    LOCAL CONST Robtarget Tr_meulage_bavure_392 := [[123.2293125,134.237953125,21.5],[0.365324878383577,-0.417802676522739,-0.626220329354095,0.547564385098326],[0,0,0,0],[8.999999E+09,8.999999E+09,8.999999E+09,8.999999E+09,8.999999E+09,8.999999E+09]];
    LOCAL CONST Robtarget Tr_meulage_bavure_393 := [[120.6318984375,139.860234375,21.5],[0.3646126685295,-0.41742546939904,-0.626882481156863,0.547569113686486],[0,0,0,0],[8.999999E+09,8.999999E+09,8.999999E+09,8.999999E+09,8.999999E+09,8.999999E+09]];
    LOCAL CONST Robtarget Tr_meulage_bavure_394 := [[119.7307734375,142.1045,21.5],[0.363803096049032,-0.416925869952999,-0.627615947970583,0.547648014807011],[0,0,0,0],[8.999999E+09,8.999999E+09,8.999999E+09,8.999999E+09,8.999999E+09,8.999999E+09]];
    LOCAL CONST Robtarget Tr_meulage_bavure_395 := [[119.108765625,144.030703125,21.5],[0.362728439124589,-0.416118032571449,-0.628549716058463,0.547904295349043],[0,0,0,0],[8.999999E+09,8.999999E+09,8.999999E+09,8.999999E+09,8.999999E+09,8.999999E+09]];
    LOCAL CONST Robtarget Tr_meulage_bavure_396 := [[118.348453125,146.077265625,21.5],[0.361294289455634,-0.414888689677899,-0.629752649770469,0.548402600004028],[0,0,0,0],[8.999999E+09,8.999999E+09,8.999999E+09,8.999999E+09,8.999999E+09,8.999999E+09]];
    LOCAL CONST Robtarget Tr_meulage_bavure_397 := [[117.2526875,148.617953125,21.5],[0.35949752433227,-0.413236866055573,-0.631224964075012,0.549137384686234],[0,0,0,0],[8.999999E+09,8.999999E+09,8.999999E+09,8.999999E+09,8.999999E+09,8.999999E+09]];
    LOCAL CONST Robtarget Tr_meulage_bavure_398 := [[116.4586171875,150.514953125,21.5],[0.357426668393585,-0.411263124366953,-0.632896063989253,0.550046717510346],[0,0,0,0],[8.999999E+09,8.999999E+09,8.999999E+09,8.999999E+09,8.999999E+09,8.999999E+09]];
    LOCAL CONST Robtarget Tr_meulage_bavure_399 := [[115.483578125,152.6576875,21.5],[0.355235316197575,-0.409147915918491,-0.634649279253162,0.55102281746676],[0,0,0,0],[8.999999E+09,8.999999E+09,8.999999E+09,8.999999E+09,8.999999E+09,8.999999E+09]];
    LOCAL CONST Robtarget Tr_meulage_bavure_400 := [[115.30321875,153.038,21.5],[0.353116300669102,-0.407109354480308,-0.636339473739805,0.551944676445876],[0,0,0,0],[8.999999E+09,8.999999E+09,8.999999E+09,8.999999E+09,8.999999E+09,8.999999E+09]];
    LOCAL CONST Robtarget Tr_meulage_bavure_401 := [[113.392453125,157.026609375,21.5],[0.351249562294065,-0.405358318756695,-0.637836707518237,0.552695859352383],[0,0,0,0],[8.999999E+09,8.999999E+09,8.999999E+09,8.999999E+09,8.999999E+09,8.999999E+09]];
    LOCAL CONST Robtarget Tr_meulage_bavure_402 := [[111.789640625,160.5481875,21.5],[0.349780045613179,-0.404061741909902,-0.639037894404603,0.553189477422075],[0,0,0,0],[8.999999E+09,8.999999E+09,8.999999E+09,8.999999E+09,8.999999E+09,8.999999E+09]];
    LOCAL CONST Robtarget Tr_meulage_bavure_403 := [[111.554078125,161.02996875,21.5],[0.348771840415515,-0.403295967871138,-0.639900183230376,0.553388038480945],[0,0,0,0],[8.999999E+09,8.999999E+09,8.999999E+09,8.999999E+09,8.999999E+09,8.999999E+09]];
    LOCAL CONST Robtarget Tr_meulage_bavure_404 := [[111.5132421875,161.124546875,21.5],[0.348208503244956,-0.403042649721828,-0.640437546956707,0.553305710454167],[0,0,0,0],[8.999999E+09,8.999999E+09,8.999999E+09,8.999999E+09,8.999999E+09,8.999999E+09]];
    LOCAL CONST Robtarget Tr_meulage_bavure_405 := [[111.45303125,161.24990625,21.5],[0.34797926768379,-0.40317690822812,-0.640731836832706,0.553011322852303],[0,0,0,0],[8.999999E+09,8.999999E+09,8.999999E+09,8.999999E+09,8.999999E+09,8.999999E+09]];
    LOCAL CONST Robtarget Tr_meulage_bavure_406 := [[109.664703125,164.673953125,21.5],[0.347911501640597,-0.40349693803522,-0.640907643054192,0.552616685503711],[0,0,0,0],[8.999999E+09,8.999999E+09,8.999999E+09,8.999999E+09,8.999999E+09,8.999999E+09]];
    LOCAL CONST Robtarget Tr_meulage_bavure_407 := [[109.3512578125,165.311765625,21.5],[0.347796802264797,-0.40375948552209,-0.641116279922809,0.552254993461587],[0,0,0,0],[8.999999E+09,8.999999E+09,8.999999E+09,8.999999E+09,8.999999E+09,8.999999E+09]];
    LOCAL CONST Robtarget Tr_meulage_bavure_408 := [[106.2381875,171.797703125,21.5],[0.347430621451574,-0.403728519395173,-0.641508118263495,0.552053059140862],[0,0,0,0],[8.999999E+09,8.999999E+09,8.999999E+09,8.999999E+09,8.999999E+09,8.999999E+09]];
    LOCAL CONST Robtarget Tr_meulage_bavure_409 := [[105.573640625,173.400671875,21.5],[0.34666342359124,-0.403226194397503,-0.64219160057769,0.552107829181196],[0,0,0,0],[8.999999E+09,8.999999E+09,8.999999E+09,8.999999E+09,8.999999E+09,8.999999E+09]];
    LOCAL CONST Robtarget Tr_meulage_bavure_410 := [[104.5446484375,175.74321875,21.5],[0.345413274544686,-0.402154478934636,-0.643224767495469,0.552470219397869],[0,0,0,0],[8.999999E+09,8.999999E+09,8.999999E+09,8.999999E+09,8.999999E+09,8.999999E+09]];
    LOCAL CONST Robtarget Tr_meulage_bavure_411 := [[103.92953125,176.899171875,21.5],[0.34368116327913,-0.400511497135502,-0.644602879657129,0.553137348410971],[0,0,0,0],[8.999999E+09,8.999999E+09,8.999999E+09,8.999999E+09,8.999999E+09,8.999999E+09]];
    LOCAL CONST Robtarget Tr_meulage_bavure_412 := [[103.241484375,178.22771875,21.5],[0.341551514127714,-0.398394425670201,-0.646259664142013,0.554051343554936],[0,0,0,0],[8.999999E+09,8.999999E+09,8.999999E+09,8.999999E+09,8.999999E+09,8.999999E+09]];
    LOCAL CONST Robtarget Tr_meulage_bavure_413 := [[102.9495859375,178.82403125,21.5],[0.339159708641225,-0.395957401256905,-0.648091582916801,0.555126768023911],[0,0,0,0],[8.999999E+09,8.999999E+09,8.999999E+09,8.999999E+09,8.999999E+09,8.999999E+09]];
    LOCAL CONST Robtarget Tr_meulage_bavure_414 := [[99.8190625,184.99203125,21.5],[0.336664877214233,-0.39338158108794,-0.649980010542665,0.556267631636098],[0,0,0,0],[8.999999E+09,8.999999E+09,8.999999E+09,8.999999E+09,8.999999E+09,8.999999E+09]];
    LOCAL CONST Robtarget Tr_meulage_bavure_415 := [[98.8109765625,186.739015625,21.5],[0.334213643527929,-0.390838206503484,-0.651820001777444,0.557384447307044],[0,0,0,0],[8.999999E+09,8.999999E+09,8.999999E+09,8.999999E+09,8.999999E+09,8.999999E+09]];
    LOCAL CONST Robtarget Tr_meulage_bavure_416 := [[96.223203125,191.122984375,21.5],[0.331906128976775,-0.388441424497442,-0.653541237438173,0.558422270553237],[0,0,0,0],[8.999999E+09,8.999999E+09,8.999999E+09,8.999999E+09,8.999999E+09,8.999999E+09]];
    LOCAL CONST Robtarget Tr_meulage_bavure_417 := [[95.8459453125,191.848875,21.5],[0.329782886774544,-0.386237077058502,-0.655116976082171,0.559362061231279],[0,0,0,0],[8.999999E+09,8.999999E+09,8.999999E+09,8.999999E+09,8.999999E+09,8.999999E+09]];
    LOCAL CONST Robtarget Tr_meulage_bavure_418 := [[92.463046875,198.07146875,21.5],[0.327832239999258,-0.384211623196163,-0.656557507184878,0.560213968745172],[0,0,0,0],[8.999999E+09,8.999999E+09,8.999999E+09,8.999999E+09,8.999999E+09,8.999999E+09]];
    LOCAL CONST Robtarget Tr_meulage_bavure_419 := [[90.7008046875,201.166375,21.5],[0.326001741527339,-0.38230075368062,-0.657899339305977,0.561014667898382],[0,0,0,0],[8.999999E+09,8.999999E+09,8.999999E+09,8.999999E+09,8.999999E+09,8.999999E+09]];
    LOCAL CONST Robtarget Tr_meulage_bavure_420 := [[89.685421875,203.134609375,21.5],[0.32421441231465,-0.380410965519129,-0.659194370838049,0.561814287479145],[0,0,0,0],[8.999999E+09,8.999999E+09,8.999999E+09,8.999999E+09,8.999999E+09,8.999999E+09]];
    LOCAL CONST Robtarget Tr_meulage_bavure_421 := [[88.7899140625,204.7486875,21.5],[0.322389107164825,-0.378447015897074,-0.660497192024121,0.562660269672843],[0,0,0,0],[8.999999E+09,8.999999E+09,8.999999E+09,8.999999E+09,8.999999E+09,8.999999E+09]];
    LOCAL CONST Robtarget Tr_meulage_bavure_422 := [[88.1928984375,205.782015625,21.5],[0.320460920439119,-0.376330604631915,-0.661849248538786,0.563591737605631],[0,0,0,0],[8.999999E+09,8.999999E+09,8.999999E+09,8.999999E+09,8.999999E+09,8.999999E+09]];
    LOCAL CONST Robtarget Tr_meulage_bavure_423 := [[87.51946875,206.94284375,21.5],[0.318384606952656,-0.374006932194033,-0.663277721464299,0.564635033393729],[0,0,0,0],[8.999999E+09,8.999999E+09,8.999999E+09,8.999999E+09,8.999999E+09,8.999999E+09]];
    LOCAL CONST Robtarget Tr_meulage_bavure_424 := [[82.9292265625,214.408875,21.5],[0.316149517900522,-0.371459858394791,-0.664784972159725,0.565798547827036],[0,0,0,0],[8.999999E+09,8.999999E+09,8.999999E+09,8.999999E+09,8.999999E+09,8.999999E+09]];
    LOCAL CONST Robtarget Tr_meulage_bavure_425 := [[82.8541875,214.52709375,21.5],[0.31376219441939,-0.368696993357463,-0.666363021379249,0.567076834459507],[0,0,0,0],[8.999999E+09,8.999999E+09,8.999999E+09,8.999999E+09,8.999999E+09,8.999999E+09]];
    LOCAL CONST Robtarget Tr_meulage_bavure_426 := [[82.726046875,214.73296875,21.5],[0.311250217448688,-0.365749884059349,-0.667989819633394,0.568453978185449],[0,0,0,0],[8.999999E+09,8.999999E+09,8.999999E+09,8.999999E+09,8.999999E+09,8.999999E+09]];
    LOCAL CONST Robtarget Tr_meulage_bavure_427 := [[77.443234375,223.1875625,21.5],[0.308652711768212,-0.362662646255843,-0.669635933625859,0.569909663829156],[0,0,0,0],[8.999999E+09,8.999999E+09,8.999999E+09,8.999999E+09,8.999999E+09,8.999999E+09]];
    LOCAL CONST Robtarget Tr_meulage_bavure_428 := [[76.0887734375,225.3150625,21.5],[0.306016386673545,-0.359491315340013,-0.671269404439817,0.571416968548702],[0,0,0,0],[8.999999E+09,8.999999E+09,8.999999E+09,8.999999E+09,8.999999E+09,8.999999E+09]];
    LOCAL CONST Robtarget Tr_meulage_bavure_429 := [[74.37640625,227.81146875,21.5],[0.303387642067638,-0.356290732601125,-0.672859367913488,0.572951240084402],[0,0,0,0],[8.999999E+09,8.999999E+09,8.999999E+09,8.999999E+09,8.999999E+09,8.999999E+09]];
    LOCAL CONST Robtarget Tr_meulage_bavure_430 := [[68.2574453125,236.729,21.5],[0.300808323404873,-0.353108038227415,-0.674377917318904,0.574494117064877],[0,0,0,0],[8.999999E+09,8.999999E+09,8.999999E+09,8.999999E+09,8.999999E+09,8.999999E+09]];
    LOCAL CONST Robtarget Tr_meulage_bavure_431 := [[67.4715,237.87903125,21.5],[0.298307331372168,-0.349979154564493,-0.675808150496031,0.576030095692119],[0,0,0,0],[8.999999E+09,8.999999E+09,8.999999E+09,8.999999E+09,8.999999E+09,8.999999E+09]];
    LOCAL CONST Robtarget Tr_meulage_bavure_432 := [[64.73254296875,241.804015625,21.5],[0.29590323329365,-0.34692572251121,-0.677139156497948,0.577552060271354],[0,0,0,0],[8.999999E+09,8.999999E+09,8.999999E+09,8.999999E+09,8.999999E+09,8.999999E+09]];
    LOCAL CONST Robtarget Tr_meulage_bavure_433 := [[64.363859375,242.338875,21.5],[0.293608347744609,-0.343964602763721,-0.678365598990462,0.579053196422045],[0,0,0,0],[8.999999E+09,8.999999E+09,8.999999E+09,8.999999E+09,8.999999E+09,8.999999E+09]];
    LOCAL CONST Robtarget Tr_meulage_bavure_434 := [[61.49722265625,246.202390625,21.5],[0.291423878540126,-0.341097438253869,-0.67948788946556,0.580534984908676],[0,0,0,0],[8.999999E+09,8.999999E+09,8.999999E+09,8.999999E+09,8.999999E+09,8.999999E+09]];
    LOCAL CONST Robtarget Tr_meulage_bavure_435 := [[61.4078671875,246.320796875,21.5],[0.289335193516394,-0.338307694283393,-0.680515840627853,0.582006220272646],[0,0,0,0],[8.999999E+09,8.999999E+09,8.999999E+09,8.999999E+09,8.999999E+09,8.999999E+09]];
    LOCAL CONST Robtarget Tr_meulage_bavure_436 := [[60.460328125,247.569390625,21.5],[0.287317708905303,-0.335572671606102,-0.681467718916006,0.583473447807153],[0,0,0,0],[8.999999E+09,8.999999E+09,8.999999E+09,8.999999E+09,8.999999E+09,8.999999E+09]];
    LOCAL CONST Robtarget Tr_meulage_bavure_437 := [[58.3609296875,250.421015625,21.5],[0.285327430113036,-0.332838804964973,-0.682367604268253,0.584962426297437],[0,0,0,0],[8.999999E+09,8.999999E+09,8.999999E+09,8.999999E+09,8.999999E+09,8.999999E+09]];
    LOCAL CONST Robtarget Tr_meulage_bavure_438 := [[56.72735546875,252.611640625,21.5],[0.283294917264907,-0.330032027158558,-0.68325802082939,0.586499213873119],[0,0,0,0],[8.999999E+09,8.999999E+09,8.999999E+09,8.999999E+09,8.999999E+09,8.999999E+09]];
    LOCAL CONST Robtarget Tr_meulage_bavure_439 := [[56.11966015625,253.3434375,21.5],[0.281118816189949,-0.327035188516629,-0.684193876122193,0.588131733995662],[0,0,0,0],[8.999999E+09,8.999999E+09,8.999999E+09,8.999999E+09,8.999999E+09,8.999999E+09]];
    LOCAL CONST Robtarget Tr_meulage_bavure_440 := [[53.942109375,255.9426875,21.5],[0.278670537913217,-0.323704550533762,-0.685244908508551,0.589913138204262],[0,0,0,0],[8.999999E+09,8.999999E+09,8.999999E+09,8.999999E+09,8.999999E+09,8.999999E+09]];
    LOCAL CONST Robtarget Tr_meulage_bavure_441 := [[52.053375,258.2940625,21.5],[0.275780385089803,-0.319847556218044,-0.686497756579809,0.591915154555071],[0,0,0,0],[8.999999E+09,8.999999E+09,8.999999E+09,8.999999E+09,8.999999E+09,8.999999E+09]];
    LOCAL CONST Robtarget Tr_meulage_bavure_442 := [[50.915984375,259.725765625,21.5],[0.272271064189163,-0.315265305626162,-0.688037190555852,0.594206259716064],[0,0,0,0],[8.999999E+09,8.999999E+09,8.999999E+09,8.999999E+09,8.999999E+09,8.999999E+09]];
    LOCAL CONST Robtarget Tr_meulage_bavure_443 := [[50.12555078125,260.70153125,21.5],[0.267918294793822,-0.309709378512022,-0.689965854732275,0.59686431245303],[0,0,0,0],[8.999999E+09,8.999999E+09,8.999999E+09,8.999999E+09,8.999999E+09,8.999999E+09]];
    LOCAL CONST Robtarget Tr_meulage_bavure_444 := [[48.66555859375,262.7159375,21.5],[0.262537588739252,-0.302972431940772,-0.692347864523534,0.599946793034662],[0,0,0,0],[8.999999E+09,8.999999E+09,8.999999E+09,8.999999E+09,8.999999E+09,8.999999E+09]];
    LOCAL CONST Robtarget Tr_meulage_bavure_445 := [[46.71563671875,264.9346875,21.5],[0.255944756105986,-0.29485466848261,-0.695235613162406,0.603490222362012],[0,0,0,0],[8.999999E+09,8.999999E+09,8.999999E+09,8.999999E+09,8.999999E+09,8.999999E+09]];
    LOCAL CONST Robtarget Tr_meulage_bavure_446 := [[46.5646953125,265.1093125,21.5],[0.247999035077578,-0.285205864760236,-0.698640894972251,0.607498965578813],[0,0,0,0],[8.999999E+09,8.999999E+09,8.999999E+09,8.999999E+09,8.999999E+09,8.999999E+09]];
    LOCAL CONST Robtarget Tr_meulage_bavure_447 := [[44.751953125,267.015625,21.5],[0.238597601740774,-0.273919505017455,-0.702538819260011,0.611946481848937],[0,0,0,0],[8.999999E+09,8.999999E+09,8.999999E+09,8.999999E+09,8.999999E+09,8.999999E+09]];
    LOCAL CONST Robtarget Tr_meulage_bavure_448 := [[43.69085546875,268.03271875,21.5],[0.22767833045319,-0.260938909430781,-0.706871806286317,0.616770389095199],[0,0,0,0],[8.999999E+09,8.999999E+09,8.999999E+09,8.999999E+09,8.999999E+09,8.999999E+09]];
    LOCAL CONST Robtarget Tr_meulage_bavure_449 := [[42.5225234375,269.16328125,21.5],[0.21513211664799,-0.246147934874376,-0.711580747640468,0.6219181667479],[0,0,0,0],[8.999999E+09,8.999999E+09,8.999999E+09,8.999999E+09,8.999999E+09,8.999999E+09]];
    LOCAL CONST Robtarget Tr_meulage_bavure_450 := [[39.8036484375,271.28553125,21.5],[0.200795358072077,-0.229372827806106,-0.716609689534343,0.627327572251076],[0,0,0,0],[8.999999E+09,8.999999E+09,8.999999E+09,8.999999E+09,8.999999E+09,8.999999E+09]];
    LOCAL CONST Robtarget Tr_meulage_bavure_451 := [[39.348265625,271.6664375,21.5],[0.184308914859871,-0.210213077062587,-0.721933668610848,0.632971140148694],[0,0,0,0],[8.999999E+09,8.999999E+09,8.999999E+09,8.999999E+09,8.999999E+09,8.999999E+09]];
    LOCAL CONST Robtarget Tr_meulage_bavure_452 := [[38.8030390625,272.0653125,21.5],[0.165142457430749,-0.188075192391745,-0.727516608940282,0.638807697571478],[0,0,0,0],[8.999999E+09,8.999999E+09,8.999999E+09,8.999999E+09,8.999999E+09,8.999999E+09]];
    LOCAL CONST Robtarget Tr_meulage_bavure_453 := [[38.28860546875,272.4004375,21.5],[0.142613659357805,-0.162194053814503,-0.733258212509643,0.644737796983361],[0,0,0,0],[8.999999E+09,8.999999E+09,8.999999E+09,8.999999E+09,8.999999E+09,8.999999E+09]];
    LOCAL CONST Robtarget Tr_meulage_bavure_454 := [[35.35888671875,274.33259375,21.5],[0.116101172092569,-0.131873584971531,-0.738889699777655,0.650516630831199],[0,0,0,0],[8.999999E+09,8.999999E+09,8.999999E+09,8.999999E+09,8.999999E+09,8.999999E+09]];
    LOCAL CONST Robtarget Tr_meulage_bavure_455 := [[32.9671953125,275.36775,21.5],[0.0854041790502875,-0.0968947501151324,-0.743904197491431,0.655685960315991],[0,0,0,0],[8.999999E+09,8.999999E+09,8.999999E+09,8.999999E+09,8.999999E+09,8.999999E+09]];
    LOCAL CONST Robtarget Tr_meulage_bavure_456 := [[32.05551171875,275.79084375,21.5],[0.0511829476564017,-0.0580099355466601,-0.747605294302051,0.659622223078193],[0,0,0,0],[8.999999E+09,8.999999E+09,8.999999E+09,8.999999E+09,8.999999E+09,8.999999E+09]];
    LOCAL CONST Robtarget Tr_meulage_bavure_457 := [[29.390564453125,276.489125,21.5],[0.0152254747357147,-0.0172411026503729,-0.749364758188975,0.661757801981095],[0,0,0,0],[8.999999E+09,8.999999E+09,8.999999E+09,8.999999E+09,8.999999E+09,8.999999E+09]];
    LOCAL CONST Robtarget Tr_meulage_bavure_458 := [[28.4075625,276.720875,21.5],[0.0195700038398143,-0.022144474819729,0.748993942157689,-0.661917450892294],[0,0,0,0],[8.999999E+09,8.999999E+09,8.999999E+09,8.999999E+09,8.999999E+09,8.999999E+09]];
    LOCAL CONST Robtarget Tr_meulage_bavure_459 := [[26.3603828125,276.49390625,21.5],[0.0500081945809172,-0.0565540862117695,0.746993014988088,-0.660531794364598],[0,0,0,0],[8.999999E+09,8.999999E+09,8.999999E+09,8.999999E+09,8.999999E+09,8.999999E+09]];
    LOCAL CONST Robtarget Tr_meulage_bavure_460 := [[25.433501953125,276.29975,21.5],[0.0733571795413084,-0.0829246680782452,0.744388584799774,-0.658504258493175],[0,0,0,0],[8.999999E+09,8.999999E+09,8.999999E+09,8.999999E+09,8.999999E+09,8.999999E+09]];
    LOCAL CONST Robtarget Tr_meulage_bavure_461 := [[24.332091796875,275.67628125,21.5],[0.0879144872089189,-0.0993550619133242,0.742288959841461,-0.656815586529792],[0,0,0,0],[8.999999E+09,8.999999E+09,8.999999E+09,8.999999E+09,8.999999E+09,8.999999E+09]];
    LOCAL CONST Robtarget Tr_meulage_bavure_462 := [[22.54901171875,274.7054375,21.5],[0.0928540392810854,-0.104928771858531,0.741494246719152,-0.656166413578023],[0,0,0,0],[8.999999E+09,8.999999E+09,8.999999E+09,8.999999E+09,8.999999E+09,8.999999E+09]];
    !
    !Declaration des points de tronconnage

    !Tronconnage_0 : Tronconnage0
    LOCAL CONST Robtarget Tronconnage_0 := [[150.06140625,-131.4606875,18.53103125],[0.0615890587455401,0.0400566245283354,0.705971293206314,0.704419468671074],[0,0,0,0],[8.999999E+09,8.999999E+09,8.999999E+09,8.999999E+09,8.999999E+09,8.999999E+09]];

    !Tronconnage_1 : Tronconnage1
    LOCAL CONST Robtarget Tronconnage_1 := [[47.56173046875,151.621203125,2.28631591796875],[0.709186160331499,-0.00109137083629826,-0.705019569723866,0.00109782072176393],[0,0,0,0],[8.999999E+09,8.999999E+09,8.999999E+09,8.999999E+09,8.999999E+09,8.999999E+09]];

    !
    !Cycle
    LOCAL PROC Cycle()
        !
        Prise;
        !
        Tronconnage;
        !
        Meulage;
        !
        !
        Depose;
        !
    ENDPROC

    !Trajectoire de prise de la pièce
    LOCAL PROC PRISE()

		!
        !Trigger localisation
        LocalisationPieceTable 702 \model:=1;
        !
        !Approche
		MoveJ Reltool(PicKPosition,0,0,-100),V1000,Z0,Tool_Prehenseur \Wobj:=Wobj_vision;
		MoveL Reltool(PicKPosition,0,0,-50),V500,Z0,Tool_Prehenseur \Wobj:=Wobj_vision;
		MoveL Reltool(PicKPosition,0,0,-10),V200,Z0,Tool_Prehenseur \Wobj:=Wobj_vision;
		MoveL PicKPosition,V100,Fine,Tool_Prehenseur \Wobj:=Wobj_vision;

        !Fermeture pince
		Gripper_Close;
        !
		MoveL Reltool(PicKPosition,0,0,-100),V500,Z0,Tool_Prehenseur \Wobj:=Wobj_vision;

        !Trigger relocalisation
		LocalisationPiecePrehenseur 702 \model:=1,Ref;
        !
        PEO;
        !
    ENDPROC

    !Trajectoire de tronconnage
    LOCAL PROC Tronconnage()
        !
        !StartMotor1();
        !
        ConfJ \Off;
        ConfL \Off;

        !Trajectoire
            !---------- tronconnage zone : 1 ------------

            !Approche PLAN

            Go_to_Tronconnage_Plan;
            Tool := ToolOffset(Tool_M2_D490_S180 \X \Z);
            !
            !Approche
            MoveJ Reltool(Tronconnage_0,0,0,-300),V1000,Z0,Tool \Wobj:=Wobj_Part_0;
            MoveL Reltool(Tronconnage_0,0,0,-200),V500,Z0,Tool \Wobj:=Wobj_Part_0;
            MoveL Reltool(Tronconnage_0,0,0,-150),V100,Z0,Tool \Wobj:=Wobj_Part_0;
            !
            Movel reltool(Tronconnage_0,0,0,-33.7070078125),VitesseTronconnageApp,Z0,Tool \Wobj:=Wobj_Part_0;
            Movel Tronconnage_0,VitesseTronconnage,Z0,Tool \Wobj:=Wobj_Part_0;
            Movel reltool(Tronconnage_0,0,0,33.7070078125),VitesseTronconnageApp,Z0,Tool \Wobj:=Wobj_Part_0;
            !
            !Degagement
            MoveL Reltool(Tronconnage_0,0,0,-150),V100,Z0,Tool \Wobj:=Wobj_Part_0;
            MoveL Reltool(Tronconnage_0,0,0,-200),V500,Z0,Tool \Wobj:=Wobj_Part_0;
            MoveJ Reltool(Tronconnage_0,0,0,-300),V1000,Z0,Tool \Wobj:=Wobj_Part_0;

            !Degagement PLAN

            Go_to_Tronconnage_Plan;
            !
            !
        !Trajectoire
            !---------- tronconnage zone : 1 ------------

            !Approche DESSOUS

            Go_to_Tronconnage_Dessous;
            Tool := ToolOffset(Tool_M2_D490_S180 \X \Z);
            !
            !Approche
            MoveJ Reltool(Tronconnage_1,0,0,-300),V1000,Z0,Tool \Wobj:=Wobj_Part_0;
            MoveL Reltool(Tronconnage_1,0,0,-200),V500,Z0,Tool \Wobj:=Wobj_Part_0;
            MoveL Reltool(Tronconnage_1,0,0,-150),V100,Z0,Tool \Wobj:=Wobj_Part_0;
            !
            Movel reltool(Tronconnage_1,0,0,-23.504642578125),VitesseTronconnageApp,Z0,Tool \Wobj:=Wobj_Part_0;
            Movel Tronconnage_1,VitesseTronconnage,Z0,Tool \Wobj:=Wobj_Part_0;
            Movel reltool(Tronconnage_1,0,0,23.504642578125),VitesseTronconnageApp,Z0,Tool \Wobj:=Wobj_Part_0;
            !
            !Degagement
            MoveL Reltool(Tronconnage_1,0,0,-150),V100,Z0,Tool \Wobj:=Wobj_Part_0;
            MoveL Reltool(Tronconnage_1,0,0,-200),V500,Z0,Tool \Wobj:=Wobj_Part_0;
            MoveJ Reltool(Tronconnage_1,0,0,-300),V1000,Z0,Tool \Wobj:=Wobj_Part_0;

            !Degagement DESSOUS

            Go_to_Tronconnage_Dessous;
            !
            !

    ENDPROC


    !Trajectoire de meulage
    LOCAL PROC Meulage()
        !
        !StartMotor2();
        !

        ConfJ \Off;
        ConfL \Off;


        !---------- Meulage zone : 1 ------------

        !Approche PLAN

        Go_to_Meulage_Plan;
		Tool := ToolOffset(Tool_M1_D500_S0 \Z);

        !
        !Approche
        MoveJ Reltool(Tr_meulage_motif_1_0,0,0,-200),V1000,Z0,Tool \Wobj:=Wobj_Part_0;
        MoveL Reltool(Tr_meulage_motif_1_0,0,0,-100),V500,Z0,Tool \Wobj:=Wobj_Part_0;
        MoveL Reltool(Tr_meulage_motif_1_0,0,0,-10),V100,Z0,Tool \Wobj:=Wobj_Part_0;
        !
        !Trajectoire
        Movel Tr_meulage_motif_1_0,VitesseLente,Z0,Tool \Wobj:=Wobj_Part_0;
        Movel Tr_meulage_motif_1_1,VitesseLente,Z0,Tool \Wobj:=Wobj_Part_0;
        Movel Tr_meulage_motif_1_2,VitesseLente,Z0,Tool \Wobj:=Wobj_Part_0;
        Movel Tr_meulage_motif_1_3,VitesseLente,Z0,Tool \Wobj:=Wobj_Part_0;
        Movel Tr_meulage_motif_1_4,VitesseLente,Z0,Tool \Wobj:=Wobj_Part_0;
        Movel Tr_meulage_motif_1_5,VitesseLente,Z0,Tool \Wobj:=Wobj_Part_0;
        Movel Tr_meulage_motif_1_6,VitesseLente,Z0,Tool \Wobj:=Wobj_Part_0;
        Movel Tr_meulage_motif_1_7,VitesseLente,Z0,Tool \Wobj:=Wobj_Part_0;
        Movel Tr_meulage_motif_1_8,VitesseLente,Z0,Tool \Wobj:=Wobj_Part_0;
        Movel Tr_meulage_motif_1_9,VitesseLente,Z0,Tool \Wobj:=Wobj_Part_0;
        Movel Tr_meulage_motif_1_10,VitesseLente,Z0,Tool \Wobj:=Wobj_Part_0;
        Movel Tr_meulage_motif_1_11,VitesseLente,Z0,Tool \Wobj:=Wobj_Part_0;
        Movel Tr_meulage_motif_1_12,VitesseLente,Z0,Tool \Wobj:=Wobj_Part_0;
        Movel Tr_meulage_motif_1_13,VitesseLente,Z0,Tool \Wobj:=Wobj_Part_0;
        Movel Tr_meulage_motif_1_14,VitesseLente,Z0,Tool \Wobj:=Wobj_Part_0;
        Movel Tr_meulage_motif_1_15,VitesseLente,Z0,Tool \Wobj:=Wobj_Part_0;
        Movel Tr_meulage_motif_1_16,VitesseLente,Z0,Tool \Wobj:=Wobj_Part_0;
        Movel Tr_meulage_motif_1_17,VitesseLente,Z0,Tool \Wobj:=Wobj_Part_0;
        Movel Tr_meulage_motif_1_18,VitesseLente,Z0,Tool \Wobj:=Wobj_Part_0;
        Movel Tr_meulage_motif_1_19,VitesseLente,Z0,Tool \Wobj:=Wobj_Part_0;
        Movel Tr_meulage_motif_1_20,VitesseLente,Z0,Tool \Wobj:=Wobj_Part_0;
        Movel Tr_meulage_motif_1_21,VitesseLente,Z0,Tool \Wobj:=Wobj_Part_0;
        Movel Tr_meulage_motif_1_22,VitesseLente,Z0,Tool \Wobj:=Wobj_Part_0;
        Movel Tr_meulage_motif_1_23,VitesseLente,Z0,Tool \Wobj:=Wobj_Part_0;
        Movel Tr_meulage_motif_1_24,VitesseLente,Z0,Tool \Wobj:=Wobj_Part_0;
        Movel Tr_meulage_motif_1_25,VitesseLente,Z0,Tool \Wobj:=Wobj_Part_0;
        Movel Tr_meulage_motif_1_26,VitesseLente,Z0,Tool \Wobj:=Wobj_Part_0;
        Movel Tr_meulage_motif_1_27,VitesseLente,Z0,Tool \Wobj:=Wobj_Part_0;
        Movel Tr_meulage_motif_1_28,VitesseLente,Z0,Tool \Wobj:=Wobj_Part_0;
        Movel Tr_meulage_motif_1_29,VitesseLente,Z0,Tool \Wobj:=Wobj_Part_0;
        Movel Tr_meulage_motif_1_30,VitesseLente,Z0,Tool \Wobj:=Wobj_Part_0;
        Movel Tr_meulage_motif_1_31,VitesseLente,Z0,Tool \Wobj:=Wobj_Part_0;
        Movel Tr_meulage_motif_1_32,VitesseLente,Z0,Tool \Wobj:=Wobj_Part_0;
        Movel Tr_meulage_motif_1_33,VitesseLente,Z0,Tool \Wobj:=Wobj_Part_0;
        Movel Tr_meulage_motif_1_34,VitesseLente,Z0,Tool \Wobj:=Wobj_Part_0;
        Movel Tr_meulage_motif_1_35,VitesseLente,Z0,Tool \Wobj:=Wobj_Part_0;
        Movel Tr_meulage_motif_1_36,VitesseLente,Z0,Tool \Wobj:=Wobj_Part_0;
        Movel Tr_meulage_motif_1_37,VitesseLente,Z0,Tool \Wobj:=Wobj_Part_0;
        Movel Tr_meulage_motif_1_38,VitesseLente,Z0,Tool \Wobj:=Wobj_Part_0;
        Movel Tr_meulage_motif_1_39,VitesseLente,Z0,Tool \Wobj:=Wobj_Part_0;
        Movel Tr_meulage_motif_1_40,VitesseLente,Z0,Tool \Wobj:=Wobj_Part_0;
        Movel Tr_meulage_motif_1_41,VitesseLente,Z0,Tool \Wobj:=Wobj_Part_0;
        Movel Tr_meulage_motif_1_42,VitesseLente,Z0,Tool \Wobj:=Wobj_Part_0;
        Movel Tr_meulage_motif_1_43,VitesseLente,Z0,Tool \Wobj:=Wobj_Part_0;
        Movel Tr_meulage_motif_1_44,VitesseLente,Z0,Tool \Wobj:=Wobj_Part_0;
        Movel Tr_meulage_motif_1_45,VitesseLente,Z0,Tool \Wobj:=Wobj_Part_0;
        Movel Tr_meulage_motif_1_46,VitesseLente,Z0,Tool \Wobj:=Wobj_Part_0;
        Movel Tr_meulage_motif_1_47,VitesseLente,Z0,Tool \Wobj:=Wobj_Part_0;
        Movel Tr_meulage_motif_1_48,VitesseLente,Z0,Tool \Wobj:=Wobj_Part_0;
        Movel Tr_meulage_motif_1_49,VitesseLente,Z0,Tool \Wobj:=Wobj_Part_0;
        Movel Tr_meulage_motif_1_50,VitesseLente,Z0,Tool \Wobj:=Wobj_Part_0;
        Movel Tr_meulage_motif_1_51,VitesseLente,Z0,Tool \Wobj:=Wobj_Part_0;
        Movel Tr_meulage_motif_1_52,VitesseLente,Z0,Tool \Wobj:=Wobj_Part_0;
        Movel Tr_meulage_motif_1_53,VitesseLente,Z0,Tool \Wobj:=Wobj_Part_0;
        Movel Tr_meulage_motif_1_54,VitesseLente,Z0,Tool \Wobj:=Wobj_Part_0;
        Movel Tr_meulage_motif_1_55,VitesseLente,Z0,Tool \Wobj:=Wobj_Part_0;
        Movel Tr_meulage_motif_1_56,VitesseLente,Z0,Tool \Wobj:=Wobj_Part_0;
        Movel Tr_meulage_motif_1_57,VitesseLente,Z0,Tool \Wobj:=Wobj_Part_0;
        Movel Tr_meulage_motif_1_58,VitesseLente,Z0,Tool \Wobj:=Wobj_Part_0;
        Movel Tr_meulage_motif_1_59,VitesseLente,Z0,Tool \Wobj:=Wobj_Part_0;
        Movel Tr_meulage_motif_1_60,VitesseLente,Z0,Tool \Wobj:=Wobj_Part_0;
        Movel Tr_meulage_motif_1_61,VitesseLente,Z0,Tool \Wobj:=Wobj_Part_0;
        Movel Tr_meulage_motif_1_62,VitesseLente,Z0,Tool \Wobj:=Wobj_Part_0;
        Movel Tr_meulage_motif_1_63,VitesseLente,Z0,Tool \Wobj:=Wobj_Part_0;
        Movel Tr_meulage_motif_1_64,VitesseLente,Z0,Tool \Wobj:=Wobj_Part_0;
        Movel Tr_meulage_motif_1_65,VitesseLente,Z0,Tool \Wobj:=Wobj_Part_0;
        Movel Tr_meulage_motif_1_66,VitesseLente,Z0,Tool \Wobj:=Wobj_Part_0;
        Movel Tr_meulage_motif_1_67,VitesseLente,Z0,Tool \Wobj:=Wobj_Part_0;
        Movel Tr_meulage_motif_1_68,VitesseLente,Z0,Tool \Wobj:=Wobj_Part_0;
        Movel Tr_meulage_motif_1_69,VitesseLente,Z0,Tool \Wobj:=Wobj_Part_0;
        Movel Tr_meulage_motif_1_70,VitesseLente,Z0,Tool \Wobj:=Wobj_Part_0;
        Movel Tr_meulage_motif_1_71,VitesseLente,Z0,Tool \Wobj:=Wobj_Part_0;
        Movel Tr_meulage_motif_1_72,VitesseLente,Z0,Tool \Wobj:=Wobj_Part_0;
        Movel Tr_meulage_motif_1_73,VitesseLente,Z0,Tool \Wobj:=Wobj_Part_0;
        Movel Tr_meulage_motif_1_74,VitesseLente,Z0,Tool \Wobj:=Wobj_Part_0;
        Movel Tr_meulage_motif_1_75,VitesseLente,Z0,Tool \Wobj:=Wobj_Part_0;
        Movel Tr_meulage_motif_1_76,VitesseLente,Z0,Tool \Wobj:=Wobj_Part_0;
        Movel Tr_meulage_motif_1_77,VitesseLente,Z0,Tool \Wobj:=Wobj_Part_0;
        Movel Tr_meulage_motif_1_78,VitesseLente,Z0,Tool \Wobj:=Wobj_Part_0;
        Movel Tr_meulage_motif_1_79,VitesseLente,Z0,Tool \Wobj:=Wobj_Part_0;
        Movel Tr_meulage_motif_1_80,VitesseLente,Z0,Tool \Wobj:=Wobj_Part_0;
        Movel Tr_meulage_motif_1_81,VitesseLente,Z0,Tool \Wobj:=Wobj_Part_0;
        Movel Tr_meulage_motif_1_82,VitesseLente,Z0,Tool \Wobj:=Wobj_Part_0;
        Movel Tr_meulage_motif_1_83,VitesseLente,Z0,Tool \Wobj:=Wobj_Part_0;
        Movel Tr_meulage_motif_1_84,VitesseLente,Z0,Tool \Wobj:=Wobj_Part_0;
        Movel Tr_meulage_motif_1_85,VitesseLente,Z0,Tool \Wobj:=Wobj_Part_0;
        Movel Tr_meulage_motif_1_86,VitesseLente,Z0,Tool \Wobj:=Wobj_Part_0;
        Movel Tr_meulage_motif_1_87,VitesseLente,Z0,Tool \Wobj:=Wobj_Part_0;
        Movel Tr_meulage_motif_1_88,VitesseLente,Z0,Tool \Wobj:=Wobj_Part_0;
        Movel Tr_meulage_motif_1_89,VitesseLente,Z0,Tool \Wobj:=Wobj_Part_0;
        Movel Tr_meulage_motif_1_90,VitesseLente,Z0,Tool \Wobj:=Wobj_Part_0;
        Movel Tr_meulage_motif_1_91,VitesseLente,Z0,Tool \Wobj:=Wobj_Part_0;
        Movel Tr_meulage_motif_1_92,VitesseLente,Z0,Tool \Wobj:=Wobj_Part_0;
        Movel Tr_meulage_motif_1_93,VitesseLente,Z0,Tool \Wobj:=Wobj_Part_0;
        Movel Tr_meulage_motif_1_94,VitesseLente,Z0,Tool \Wobj:=Wobj_Part_0;
        Movel Tr_meulage_motif_1_95,VitesseLente,Z0,Tool \Wobj:=Wobj_Part_0;
        Movel Tr_meulage_motif_1_96,VitesseLente,Z0,Tool \Wobj:=Wobj_Part_0;
        Movel Tr_meulage_motif_1_97,VitesseLente,Z0,Tool \Wobj:=Wobj_Part_0;
        Movel Tr_meulage_motif_1_98,VitesseLente,Z0,Tool \Wobj:=Wobj_Part_0;
        Movel Tr_meulage_motif_1_99,VitesseLente,Z0,Tool \Wobj:=Wobj_Part_0;
        Movel Tr_meulage_motif_1_100,VitesseLente,Z0,Tool \Wobj:=Wobj_Part_0;
        Movel Tr_meulage_motif_1_101,VitesseLente,Z0,Tool \Wobj:=Wobj_Part_0;
        Movel Tr_meulage_motif_1_102,VitesseLente,Z0,Tool \Wobj:=Wobj_Part_0;
        Movel Tr_meulage_motif_1_103,VitesseLente,Z0,Tool \Wobj:=Wobj_Part_0;
        Movel Tr_meulage_motif_1_104,VitesseLente,Z0,Tool \Wobj:=Wobj_Part_0;
        Movel Tr_meulage_motif_1_105,VitesseLente,Z0,Tool \Wobj:=Wobj_Part_0;
        Movel Tr_meulage_motif_1_106,VitesseLente,Z0,Tool \Wobj:=Wobj_Part_0;
        Movel Tr_meulage_motif_1_107,VitesseLente,Z0,Tool \Wobj:=Wobj_Part_0;
        Movel Tr_meulage_motif_1_108,VitesseLente,Z0,Tool \Wobj:=Wobj_Part_0;
        Movel Tr_meulage_motif_1_109,VitesseLente,Z0,Tool \Wobj:=Wobj_Part_0;
        Movel Tr_meulage_motif_1_110,VitesseLente,Z0,Tool \Wobj:=Wobj_Part_0;
        Movel Tr_meulage_motif_1_111,VitesseLente,Z0,Tool \Wobj:=Wobj_Part_0;
        Movel Tr_meulage_motif_1_112,VitesseLente,Z0,Tool \Wobj:=Wobj_Part_0;
        Movel Tr_meulage_motif_1_113,VitesseLente,Z0,Tool \Wobj:=Wobj_Part_0;
        Movel Tr_meulage_motif_1_114,VitesseLente,Z0,Tool \Wobj:=Wobj_Part_0;
        Movel Tr_meulage_motif_1_115,VitesseLente,Z0,Tool \Wobj:=Wobj_Part_0;
        !
        !Degagement
        MoveL Reltool(Tr_meulage_motif_1_115,0,0,-10),V100,Z0,Tool \Wobj:=Wobj_Part_0;
        MoveL Reltool(Tr_meulage_motif_1_115,0,0,-100),V500,Z0,Tool \Wobj:=Wobj_Part_0;
        MoveJ Reltool(Tr_meulage_motif_1_115,0,0,-200),V1000,Z0,Tool \Wobj:=Wobj_Part_0;


        Go_to_Meulage_Plan;
        !
        !

        !---------- Meulage zone : 2 ------------

        !Approche DESSOUS

        Go_to_Meulage_Dessous;
		Tool := ToolOffset(Tool_M1_D500_S270 \Z);
        !
        !Approche
        MoveJ Reltool(Tr_meulage_motif_2_0,0,0,-200),V1000,Z0,Tool \Wobj:=Wobj_Part_0;
        MoveL Reltool(Tr_meulage_motif_2_0,0,0,-100),V500,Z0,Tool \Wobj:=Wobj_Part_0;
        MoveL Reltool(Tr_meulage_motif_2_0,0,0,-10),V100,Z0,Tool \Wobj:=Wobj_Part_0;
        !
        !Trajectoire
        Movel Tr_meulage_motif_2_0,VitesseLente,Z0,Tool \Wobj:=Wobj_Part_0;
        Movel Tr_meulage_motif_2_1,VitesseLente,Z0,Tool \Wobj:=Wobj_Part_0;
        Movel Tr_meulage_motif_2_2,VitesseLente,Z0,Tool \Wobj:=Wobj_Part_0;
        Movel Tr_meulage_motif_2_3,VitesseLente,Z0,Tool \Wobj:=Wobj_Part_0;
        Movel Tr_meulage_motif_2_4,VitesseLente,Z0,Tool \Wobj:=Wobj_Part_0;
        Movel Tr_meulage_motif_2_5,VitesseLente,Z0,Tool \Wobj:=Wobj_Part_0;
        Movel Tr_meulage_motif_2_6,VitesseLente,Z0,Tool \Wobj:=Wobj_Part_0;
        Movel Tr_meulage_motif_2_7,VitesseLente,Z0,Tool \Wobj:=Wobj_Part_0;
        Movel Tr_meulage_motif_2_8,VitesseLente,Z0,Tool \Wobj:=Wobj_Part_0;
        Movel Tr_meulage_motif_2_9,VitesseLente,Z0,Tool \Wobj:=Wobj_Part_0;
        Movel Tr_meulage_motif_2_10,VitesseLente,Z0,Tool \Wobj:=Wobj_Part_0;
        Movel Tr_meulage_motif_2_11,VitesseLente,Z0,Tool \Wobj:=Wobj_Part_0;
        Movel Tr_meulage_motif_2_12,VitesseLente,Z0,Tool \Wobj:=Wobj_Part_0;
        Movel Tr_meulage_motif_2_13,VitesseLente,Z0,Tool \Wobj:=Wobj_Part_0;
        Movel Tr_meulage_motif_2_14,VitesseLente,Z0,Tool \Wobj:=Wobj_Part_0;
        Movel Tr_meulage_motif_2_15,VitesseLente,Z0,Tool \Wobj:=Wobj_Part_0;
        Movel Tr_meulage_motif_2_16,VitesseLente,Z0,Tool \Wobj:=Wobj_Part_0;
        Movel Tr_meulage_motif_2_17,VitesseLente,Z0,Tool \Wobj:=Wobj_Part_0;
        Movel Tr_meulage_motif_2_18,VitesseLente,Z0,Tool \Wobj:=Wobj_Part_0;
        Movel Tr_meulage_motif_2_19,VitesseLente,Z0,Tool \Wobj:=Wobj_Part_0;
        Movel Tr_meulage_motif_2_20,VitesseLente,Z0,Tool \Wobj:=Wobj_Part_0;
        Movel Tr_meulage_motif_2_21,VitesseLente,Z0,Tool \Wobj:=Wobj_Part_0;
        Movel Tr_meulage_motif_2_22,VitesseLente,Z0,Tool \Wobj:=Wobj_Part_0;
        Movel Tr_meulage_motif_2_23,VitesseLente,Z0,Tool \Wobj:=Wobj_Part_0;
        Movel Tr_meulage_motif_2_24,VitesseLente,Z0,Tool \Wobj:=Wobj_Part_0;
        Movel Tr_meulage_motif_2_25,VitesseLente,Z0,Tool \Wobj:=Wobj_Part_0;
        Movel Tr_meulage_motif_2_26,VitesseLente,Z0,Tool \Wobj:=Wobj_Part_0;
        Movel Tr_meulage_motif_2_27,VitesseLente,Z0,Tool \Wobj:=Wobj_Part_0;
        Movel Tr_meulage_motif_2_28,VitesseLente,Z0,Tool \Wobj:=Wobj_Part_0;
        Movel Tr_meulage_motif_2_29,VitesseLente,Z0,Tool \Wobj:=Wobj_Part_0;
        Movel Tr_meulage_motif_2_30,VitesseLente,Z0,Tool \Wobj:=Wobj_Part_0;
        Movel Tr_meulage_motif_2_31,VitesseLente,Z0,Tool \Wobj:=Wobj_Part_0;
        Movel Tr_meulage_motif_2_32,VitesseLente,Z0,Tool \Wobj:=Wobj_Part_0;
        Movel Tr_meulage_motif_2_33,VitesseLente,Z0,Tool \Wobj:=Wobj_Part_0;
        Movel Tr_meulage_motif_2_34,VitesseLente,Z0,Tool \Wobj:=Wobj_Part_0;
        Movel Tr_meulage_motif_2_35,VitesseLente,Z0,Tool \Wobj:=Wobj_Part_0;
        Movel Tr_meulage_motif_2_36,VitesseLente,Z0,Tool \Wobj:=Wobj_Part_0;
        Movel Tr_meulage_motif_2_37,VitesseLente,Z0,Tool \Wobj:=Wobj_Part_0;
        Movel Tr_meulage_motif_2_38,VitesseLente,Z0,Tool \Wobj:=Wobj_Part_0;
        Movel Tr_meulage_motif_2_39,VitesseLente,Z0,Tool \Wobj:=Wobj_Part_0;
        Movel Tr_meulage_motif_2_40,VitesseLente,Z0,Tool \Wobj:=Wobj_Part_0;
        Movel Tr_meulage_motif_2_41,VitesseLente,Z0,Tool \Wobj:=Wobj_Part_0;
        Movel Tr_meulage_motif_2_42,VitesseLente,Z0,Tool \Wobj:=Wobj_Part_0;
        Movel Tr_meulage_motif_2_43,VitesseLente,Z0,Tool \Wobj:=Wobj_Part_0;
        Movel Tr_meulage_motif_2_44,VitesseLente,Z0,Tool \Wobj:=Wobj_Part_0;
        Movel Tr_meulage_motif_2_45,VitesseLente,Z0,Tool \Wobj:=Wobj_Part_0;
        Movel Tr_meulage_motif_2_46,VitesseLente,Z0,Tool \Wobj:=Wobj_Part_0;
        Movel Tr_meulage_motif_2_47,VitesseLente,Z0,Tool \Wobj:=Wobj_Part_0;
        Movel Tr_meulage_motif_2_48,VitesseLente,Z0,Tool \Wobj:=Wobj_Part_0;
        Movel Tr_meulage_motif_2_49,VitesseLente,Z0,Tool \Wobj:=Wobj_Part_0;
        Movel Tr_meulage_motif_2_50,VitesseLente,Z0,Tool \Wobj:=Wobj_Part_0;
        Movel Tr_meulage_motif_2_51,VitesseLente,Z0,Tool \Wobj:=Wobj_Part_0;
        Movel Tr_meulage_motif_2_52,VitesseLente,Z0,Tool \Wobj:=Wobj_Part_0;
        Movel Tr_meulage_motif_2_53,VitesseLente,Z0,Tool \Wobj:=Wobj_Part_0;
        Movel Tr_meulage_motif_2_54,VitesseLente,Z0,Tool \Wobj:=Wobj_Part_0;
        Movel Tr_meulage_motif_2_55,VitesseLente,Z0,Tool \Wobj:=Wobj_Part_0;
        Movel Tr_meulage_motif_2_56,VitesseLente,Z0,Tool \Wobj:=Wobj_Part_0;
        Movel Tr_meulage_motif_2_57,VitesseLente,Z0,Tool \Wobj:=Wobj_Part_0;
        Movel Tr_meulage_motif_2_58,VitesseLente,Z0,Tool \Wobj:=Wobj_Part_0;
        Movel Tr_meulage_motif_2_59,VitesseLente,Z0,Tool \Wobj:=Wobj_Part_0;
        Movel Tr_meulage_motif_2_60,VitesseLente,Z0,Tool \Wobj:=Wobj_Part_0;
        Movel Tr_meulage_motif_2_61,VitesseLente,Z0,Tool \Wobj:=Wobj_Part_0;
        Movel Tr_meulage_motif_2_62,VitesseLente,Z0,Tool \Wobj:=Wobj_Part_0;
        Movel Tr_meulage_motif_2_63,VitesseLente,Z0,Tool \Wobj:=Wobj_Part_0;
        Movel Tr_meulage_motif_2_64,VitesseLente,Z0,Tool \Wobj:=Wobj_Part_0;
        Movel Tr_meulage_motif_2_65,VitesseLente,Z0,Tool \Wobj:=Wobj_Part_0;
        Movel Tr_meulage_motif_2_66,VitesseLente,Z0,Tool \Wobj:=Wobj_Part_0;
        Movel Tr_meulage_motif_2_67,VitesseLente,Z0,Tool \Wobj:=Wobj_Part_0;
        Movel Tr_meulage_motif_2_68,VitesseLente,Z0,Tool \Wobj:=Wobj_Part_0;
        Movel Tr_meulage_motif_2_69,VitesseLente,Z0,Tool \Wobj:=Wobj_Part_0;
        Movel Tr_meulage_motif_2_70,VitesseLente,Z0,Tool \Wobj:=Wobj_Part_0;
        Movel Tr_meulage_motif_2_71,VitesseLente,Z0,Tool \Wobj:=Wobj_Part_0;
        Movel Tr_meulage_motif_2_72,VitesseLente,Z0,Tool \Wobj:=Wobj_Part_0;
        Movel Tr_meulage_motif_2_73,VitesseLente,Z0,Tool \Wobj:=Wobj_Part_0;
        Movel Tr_meulage_motif_2_74,VitesseLente,Z0,Tool \Wobj:=Wobj_Part_0;
        Movel Tr_meulage_motif_2_75,VitesseLente,Z0,Tool \Wobj:=Wobj_Part_0;
        Movel Tr_meulage_motif_2_76,VitesseLente,Z0,Tool \Wobj:=Wobj_Part_0;
        Movel Tr_meulage_motif_2_77,VitesseLente,Z0,Tool \Wobj:=Wobj_Part_0;
        Movel Tr_meulage_motif_2_78,VitesseLente,Z0,Tool \Wobj:=Wobj_Part_0;
        Movel Tr_meulage_motif_2_79,VitesseLente,Z0,Tool \Wobj:=Wobj_Part_0;
        Movel Tr_meulage_motif_2_80,VitesseLente,Z0,Tool \Wobj:=Wobj_Part_0;
        Movel Tr_meulage_motif_2_81,VitesseLente,Z0,Tool \Wobj:=Wobj_Part_0;
        Movel Tr_meulage_motif_2_82,VitesseLente,Z0,Tool \Wobj:=Wobj_Part_0;
        Movel Tr_meulage_motif_2_83,VitesseLente,Z0,Tool \Wobj:=Wobj_Part_0;
        Movel Tr_meulage_motif_2_84,VitesseLente,Z0,Tool \Wobj:=Wobj_Part_0;
        Movel Tr_meulage_motif_2_85,VitesseLente,Z0,Tool \Wobj:=Wobj_Part_0;
        Movel Tr_meulage_motif_2_86,VitesseLente,Z0,Tool \Wobj:=Wobj_Part_0;
        Movel Tr_meulage_motif_2_87,VitesseLente,Z0,Tool \Wobj:=Wobj_Part_0;
        Movel Tr_meulage_motif_2_88,VitesseLente,Z0,Tool \Wobj:=Wobj_Part_0;
        Movel Tr_meulage_motif_2_89,VitesseLente,Z0,Tool \Wobj:=Wobj_Part_0;
        Movel Tr_meulage_motif_2_90,VitesseLente,Z0,Tool \Wobj:=Wobj_Part_0;
        Movel Tr_meulage_motif_2_91,VitesseLente,Z0,Tool \Wobj:=Wobj_Part_0;
        Movel Tr_meulage_motif_2_92,VitesseLente,Z0,Tool \Wobj:=Wobj_Part_0;
        Movel Tr_meulage_motif_2_93,VitesseLente,Z0,Tool \Wobj:=Wobj_Part_0;
        Movel Tr_meulage_motif_2_94,VitesseLente,Z0,Tool \Wobj:=Wobj_Part_0;
        Movel Tr_meulage_motif_2_95,VitesseLente,Z0,Tool \Wobj:=Wobj_Part_0;
        Movel Tr_meulage_motif_2_96,VitesseLente,Z0,Tool \Wobj:=Wobj_Part_0;
        Movel Tr_meulage_motif_2_97,VitesseLente,Z0,Tool \Wobj:=Wobj_Part_0;
        Movel Tr_meulage_motif_2_98,VitesseLente,Z0,Tool \Wobj:=Wobj_Part_0;
        Movel Tr_meulage_motif_2_99,VitesseLente,Z0,Tool \Wobj:=Wobj_Part_0;
        Movel Tr_meulage_motif_2_100,VitesseLente,Z0,Tool \Wobj:=Wobj_Part_0;
        Movel Tr_meulage_motif_2_101,VitesseLente,Z0,Tool \Wobj:=Wobj_Part_0;
        Movel Tr_meulage_motif_2_102,VitesseLente,Z0,Tool \Wobj:=Wobj_Part_0;
        Movel Tr_meulage_motif_2_103,VitesseLente,Z0,Tool \Wobj:=Wobj_Part_0;
        Movel Tr_meulage_motif_2_104,VitesseLente,Z0,Tool \Wobj:=Wobj_Part_0;
        Movel Tr_meulage_motif_2_105,VitesseLente,Z0,Tool \Wobj:=Wobj_Part_0;
        Movel Tr_meulage_motif_2_106,VitesseLente,Z0,Tool \Wobj:=Wobj_Part_0;
        Movel Tr_meulage_motif_2_107,VitesseLente,Z0,Tool \Wobj:=Wobj_Part_0;
        Movel Tr_meulage_motif_2_108,VitesseLente,Z0,Tool \Wobj:=Wobj_Part_0;
        Movel Tr_meulage_motif_2_109,VitesseLente,Z0,Tool \Wobj:=Wobj_Part_0;
        Movel Tr_meulage_motif_2_110,VitesseLente,Z0,Tool \Wobj:=Wobj_Part_0;
        Movel Tr_meulage_motif_2_111,VitesseLente,Z0,Tool \Wobj:=Wobj_Part_0;
        Movel Tr_meulage_motif_2_112,VitesseLente,Z0,Tool \Wobj:=Wobj_Part_0;
        Movel Tr_meulage_motif_2_113,VitesseLente,Z0,Tool \Wobj:=Wobj_Part_0;
        Movel Tr_meulage_motif_2_114,VitesseLente,Z0,Tool \Wobj:=Wobj_Part_0;
        Movel Tr_meulage_motif_2_115,VitesseLente,Z0,Tool \Wobj:=Wobj_Part_0;
        !
        !Degagement
        MoveL Reltool(Tr_meulage_motif_2_115,0,0,-10),V100,Z0,Tool \Wobj:=Wobj_Part_0;
        MoveL Reltool(Tr_meulage_motif_2_115,0,0,-100),V500,Z0,Tool \Wobj:=Wobj_Part_0;
        MoveJ Reltool(Tr_meulage_motif_2_115,0,0,-200),V1000,Z0,Tool \Wobj:=Wobj_Part_0;


        Go_to_Meulage_Dessous;
        !
        !

        !---------- Meulage zone : 3 ------------

        !Approche PLAN

        Go_to_Meulage_Plan;
		Tool := ToolOffset(Tool_M1_D500_S0 \Z);

        !
        !Approche
        MoveJ Reltool(Tr_meulage_bavure_0,0,0,-200),V1000,Z0,Tool \Wobj:=Wobj_Part_0;
        MoveL Reltool(Tr_meulage_bavure_0,0,0,-100),V500,Z0,Tool \Wobj:=Wobj_Part_0;
        MoveL Reltool(Tr_meulage_bavure_0,0,0,-10),V100,Z0,Tool \Wobj:=Wobj_Part_0;
        !
        !Trajectoire
        Movel Tr_meulage_bavure_0,VitesseRapide,Z0,Tool \Wobj:=Wobj_Part_0;
        Movel Tr_meulage_bavure_1,VitesseRapide,Z0,Tool \Wobj:=Wobj_Part_0;
        Movel Tr_meulage_bavure_2,VitesseRapide,Z0,Tool \Wobj:=Wobj_Part_0;
        Movel Tr_meulage_bavure_3,VitesseRapide,Z0,Tool \Wobj:=Wobj_Part_0;
        Movel Tr_meulage_bavure_4,VitesseRapide,Z0,Tool \Wobj:=Wobj_Part_0;
        Movel Tr_meulage_bavure_5,VitesseRapide,Z0,Tool \Wobj:=Wobj_Part_0;
        Movel Tr_meulage_bavure_6,VitesseRapide,Z0,Tool \Wobj:=Wobj_Part_0;
        Movel Tr_meulage_bavure_7,VitesseRapide,Z0,Tool \Wobj:=Wobj_Part_0;
        Movel Tr_meulage_bavure_8,VitesseRapide,Z0,Tool \Wobj:=Wobj_Part_0;
        Movel Tr_meulage_bavure_9,VitesseRapide,Z0,Tool \Wobj:=Wobj_Part_0;
        Movel Tr_meulage_bavure_10,VitesseRapide,Z0,Tool \Wobj:=Wobj_Part_0;
        Movel Tr_meulage_bavure_11,VitesseRapide,Z0,Tool \Wobj:=Wobj_Part_0;
        Movel Tr_meulage_bavure_12,VitesseRapide,Z0,Tool \Wobj:=Wobj_Part_0;
        Movel Tr_meulage_bavure_13,VitesseRapide,Z0,Tool \Wobj:=Wobj_Part_0;
        Movel Tr_meulage_bavure_14,VitesseRapide,Z0,Tool \Wobj:=Wobj_Part_0;
        Movel Tr_meulage_bavure_15,VitesseRapide,Z0,Tool \Wobj:=Wobj_Part_0;
        Movel Tr_meulage_bavure_16,VitesseRapide,Z0,Tool \Wobj:=Wobj_Part_0;
        Movel Tr_meulage_bavure_17,VitesseRapide,Z0,Tool \Wobj:=Wobj_Part_0;
        Movel Tr_meulage_bavure_18,VitesseRapide,Z0,Tool \Wobj:=Wobj_Part_0;
        Movel Tr_meulage_bavure_19,VitesseRapide,Z0,Tool \Wobj:=Wobj_Part_0;
        Movel Tr_meulage_bavure_20,VitesseRapide,Z0,Tool \Wobj:=Wobj_Part_0;
        Movel Tr_meulage_bavure_21,VitesseRapide,Z0,Tool \Wobj:=Wobj_Part_0;
        Movel Tr_meulage_bavure_22,VitesseRapide,Z0,Tool \Wobj:=Wobj_Part_0;
        Movel Tr_meulage_bavure_23,VitesseRapide,Z0,Tool \Wobj:=Wobj_Part_0;
        Movel Tr_meulage_bavure_24,VitesseRapide,Z0,Tool \Wobj:=Wobj_Part_0;
        Movel Tr_meulage_bavure_25,VitesseRapide,Z0,Tool \Wobj:=Wobj_Part_0;
        Movel Tr_meulage_bavure_26,VitesseRapide,Z0,Tool \Wobj:=Wobj_Part_0;
        Movel Tr_meulage_bavure_27,VitesseRapide,Z0,Tool \Wobj:=Wobj_Part_0;
        Movel Tr_meulage_bavure_28,VitesseRapide,Z0,Tool \Wobj:=Wobj_Part_0;
        Movel Tr_meulage_bavure_29,VitesseRapide,Z0,Tool \Wobj:=Wobj_Part_0;
        Movel Tr_meulage_bavure_30,VitesseRapide,Z0,Tool \Wobj:=Wobj_Part_0;
        Movel Tr_meulage_bavure_31,VitesseRapide,Z0,Tool \Wobj:=Wobj_Part_0;
        Movel Tr_meulage_bavure_32,VitesseRapide,Z0,Tool \Wobj:=Wobj_Part_0;
        Movel Tr_meulage_bavure_33,VitesseRapide,Z0,Tool \Wobj:=Wobj_Part_0;
        Movel Tr_meulage_bavure_34,VitesseRapide,Z0,Tool \Wobj:=Wobj_Part_0;
        Movel Tr_meulage_bavure_35,VitesseRapide,Z0,Tool \Wobj:=Wobj_Part_0;
        Movel Tr_meulage_bavure_36,VitesseRapide,Z0,Tool \Wobj:=Wobj_Part_0;
        Movel Tr_meulage_bavure_37,VitesseRapide,Z0,Tool \Wobj:=Wobj_Part_0;
        Movel Tr_meulage_bavure_38,VitesseRapide,Z0,Tool \Wobj:=Wobj_Part_0;
        Movel Tr_meulage_bavure_39,VitesseRapide,Z0,Tool \Wobj:=Wobj_Part_0;
        Movel Tr_meulage_bavure_40,VitesseRapide,Z0,Tool \Wobj:=Wobj_Part_0;
        Movel Tr_meulage_bavure_41,VitesseRapide,Z0,Tool \Wobj:=Wobj_Part_0;
        Movel Tr_meulage_bavure_42,VitesseRapide,Z0,Tool \Wobj:=Wobj_Part_0;
        Movel Tr_meulage_bavure_43,VitesseRapide,Z0,Tool \Wobj:=Wobj_Part_0;
        Movel Tr_meulage_bavure_44,VitesseRapide,Z0,Tool \Wobj:=Wobj_Part_0;
        Movel Tr_meulage_bavure_45,VitesseRapide,Z0,Tool \Wobj:=Wobj_Part_0;
        Movel Tr_meulage_bavure_46,VitesseRapide,Z0,Tool \Wobj:=Wobj_Part_0;
        Movel Tr_meulage_bavure_47,VitesseRapide,Z0,Tool \Wobj:=Wobj_Part_0;
        Movel Tr_meulage_bavure_48,VitesseRapide,Z0,Tool \Wobj:=Wobj_Part_0;
        Movel Tr_meulage_bavure_49,VitesseRapide,Z0,Tool \Wobj:=Wobj_Part_0;
        Movel Tr_meulage_bavure_50,VitesseRapide,Z0,Tool \Wobj:=Wobj_Part_0;
        Movel Tr_meulage_bavure_51,VitesseRapide,Z0,Tool \Wobj:=Wobj_Part_0;
        Movel Tr_meulage_bavure_52,VitesseRapide,Z0,Tool \Wobj:=Wobj_Part_0;
        Movel Tr_meulage_bavure_53,VitesseRapide,Z0,Tool \Wobj:=Wobj_Part_0;
        Movel Tr_meulage_bavure_54,VitesseRapide,Z0,Tool \Wobj:=Wobj_Part_0;
        Movel Tr_meulage_bavure_55,VitesseRapide,Z0,Tool \Wobj:=Wobj_Part_0;
        Movel Tr_meulage_bavure_56,VitesseRapide,Z0,Tool \Wobj:=Wobj_Part_0;
        Movel Tr_meulage_bavure_57,VitesseRapide,Z0,Tool \Wobj:=Wobj_Part_0;
        Movel Tr_meulage_bavure_58,VitesseRapide,Z0,Tool \Wobj:=Wobj_Part_0;
        Movel Tr_meulage_bavure_59,VitesseRapide,Z0,Tool \Wobj:=Wobj_Part_0;
        Movel Tr_meulage_bavure_60,VitesseRapide,Z0,Tool \Wobj:=Wobj_Part_0;
        Movel Tr_meulage_bavure_61,VitesseRapide,Z0,Tool \Wobj:=Wobj_Part_0;
        Movel Tr_meulage_bavure_62,VitesseRapide,Z0,Tool \Wobj:=Wobj_Part_0;
        Movel Tr_meulage_bavure_63,VitesseRapide,Z0,Tool \Wobj:=Wobj_Part_0;
        Movel Tr_meulage_bavure_64,VitesseRapide,Z0,Tool \Wobj:=Wobj_Part_0;
        Movel Tr_meulage_bavure_65,VitesseRapide,Z0,Tool \Wobj:=Wobj_Part_0;
        Movel Tr_meulage_bavure_66,VitesseRapide,Z0,Tool \Wobj:=Wobj_Part_0;
        Movel Tr_meulage_bavure_67,VitesseRapide,Z0,Tool \Wobj:=Wobj_Part_0;
        Movel Tr_meulage_bavure_68,VitesseRapide,Z0,Tool \Wobj:=Wobj_Part_0;
        Movel Tr_meulage_bavure_69,VitesseRapide,Z0,Tool \Wobj:=Wobj_Part_0;
        Movel Tr_meulage_bavure_70,VitesseRapide,Z0,Tool \Wobj:=Wobj_Part_0;
        Movel Tr_meulage_bavure_71,VitesseRapide,Z0,Tool \Wobj:=Wobj_Part_0;
        Movel Tr_meulage_bavure_72,VitesseRapide,Z0,Tool \Wobj:=Wobj_Part_0;
        Movel Tr_meulage_bavure_73,VitesseRapide,Z0,Tool \Wobj:=Wobj_Part_0;
        Movel Tr_meulage_bavure_74,VitesseRapide,Z0,Tool \Wobj:=Wobj_Part_0;
        Movel Tr_meulage_bavure_75,VitesseRapide,Z0,Tool \Wobj:=Wobj_Part_0;
        Movel Tr_meulage_bavure_76,VitesseRapide,Z0,Tool \Wobj:=Wobj_Part_0;
        Movel Tr_meulage_bavure_77,VitesseRapide,Z0,Tool \Wobj:=Wobj_Part_0;
        Movel Tr_meulage_bavure_78,VitesseRapide,Z0,Tool \Wobj:=Wobj_Part_0;
        Movel Tr_meulage_bavure_79,VitesseRapide,Z0,Tool \Wobj:=Wobj_Part_0;
        Movel Tr_meulage_bavure_80,VitesseRapide,Z0,Tool \Wobj:=Wobj_Part_0;
        Movel Tr_meulage_bavure_81,VitesseRapide,Z0,Tool \Wobj:=Wobj_Part_0;
        Movel Tr_meulage_bavure_82,VitesseRapide,Z0,Tool \Wobj:=Wobj_Part_0;
        Movel Tr_meulage_bavure_83,VitesseRapide,Z0,Tool \Wobj:=Wobj_Part_0;
        Movel Tr_meulage_bavure_84,VitesseRapide,Z0,Tool \Wobj:=Wobj_Part_0;
        Movel Tr_meulage_bavure_85,VitesseRapide,Z0,Tool \Wobj:=Wobj_Part_0;
        Movel Tr_meulage_bavure_86,VitesseRapide,Z0,Tool \Wobj:=Wobj_Part_0;
        Movel Tr_meulage_bavure_87,VitesseRapide,Z0,Tool \Wobj:=Wobj_Part_0;
        Movel Tr_meulage_bavure_88,VitesseRapide,Z0,Tool \Wobj:=Wobj_Part_0;
        Movel Tr_meulage_bavure_89,VitesseRapide,Z0,Tool \Wobj:=Wobj_Part_0;
        Movel Tr_meulage_bavure_90,VitesseRapide,Z0,Tool \Wobj:=Wobj_Part_0;
        Movel Tr_meulage_bavure_91,VitesseRapide,Z0,Tool \Wobj:=Wobj_Part_0;
        Movel Tr_meulage_bavure_92,VitesseRapide,Z0,Tool \Wobj:=Wobj_Part_0;
        Movel Tr_meulage_bavure_93,VitesseRapide,Z0,Tool \Wobj:=Wobj_Part_0;
        Movel Tr_meulage_bavure_94,VitesseRapide,Z0,Tool \Wobj:=Wobj_Part_0;
        Movel Tr_meulage_bavure_95,VitesseRapide,Z0,Tool \Wobj:=Wobj_Part_0;
        Movel Tr_meulage_bavure_96,VitesseRapide,Z0,Tool \Wobj:=Wobj_Part_0;
        Movel Tr_meulage_bavure_97,VitesseRapide,Z0,Tool \Wobj:=Wobj_Part_0;
        Movel Tr_meulage_bavure_98,VitesseRapide,Z0,Tool \Wobj:=Wobj_Part_0;
        Movel Tr_meulage_bavure_99,VitesseRapide,Z0,Tool \Wobj:=Wobj_Part_0;
        Movel Tr_meulage_bavure_100,VitesseRapide,Z0,Tool \Wobj:=Wobj_Part_0;
        Movel Tr_meulage_bavure_101,VitesseRapide,Z0,Tool \Wobj:=Wobj_Part_0;
        Movel Tr_meulage_bavure_102,VitesseRapide,Z0,Tool \Wobj:=Wobj_Part_0;
        Movel Tr_meulage_bavure_103,VitesseRapide,Z0,Tool \Wobj:=Wobj_Part_0;
        Movel Tr_meulage_bavure_104,VitesseRapide,Z0,Tool \Wobj:=Wobj_Part_0;
        Movel Tr_meulage_bavure_105,VitesseRapide,Z0,Tool \Wobj:=Wobj_Part_0;
        Movel Tr_meulage_bavure_106,VitesseRapide,Z0,Tool \Wobj:=Wobj_Part_0;
        Movel Tr_meulage_bavure_107,VitesseRapide,Z0,Tool \Wobj:=Wobj_Part_0;
        Movel Tr_meulage_bavure_108,VitesseRapide,Z0,Tool \Wobj:=Wobj_Part_0;
        Movel Tr_meulage_bavure_109,VitesseRapide,Z0,Tool \Wobj:=Wobj_Part_0;
        Movel Tr_meulage_bavure_110,VitesseRapide,Z0,Tool \Wobj:=Wobj_Part_0;
        Movel Tr_meulage_bavure_111,VitesseRapide,Z0,Tool \Wobj:=Wobj_Part_0;
        Movel Tr_meulage_bavure_112,VitesseRapide,Z0,Tool \Wobj:=Wobj_Part_0;
        Movel Tr_meulage_bavure_113,VitesseRapide,Z0,Tool \Wobj:=Wobj_Part_0;
        Movel Tr_meulage_bavure_114,VitesseRapide,Z0,Tool \Wobj:=Wobj_Part_0;
        Movel Tr_meulage_bavure_115,VitesseRapide,Z0,Tool \Wobj:=Wobj_Part_0;
        Movel Tr_meulage_bavure_116,VitesseRapide,Z0,Tool \Wobj:=Wobj_Part_0;
        Movel Tr_meulage_bavure_117,VitesseRapide,Z0,Tool \Wobj:=Wobj_Part_0;
        Movel Tr_meulage_bavure_118,VitesseRapide,Z0,Tool \Wobj:=Wobj_Part_0;
        Movel Tr_meulage_bavure_119,VitesseRapide,Z0,Tool \Wobj:=Wobj_Part_0;
        Movel Tr_meulage_bavure_120,VitesseRapide,Z0,Tool \Wobj:=Wobj_Part_0;
        Movel Tr_meulage_bavure_121,VitesseRapide,Z0,Tool \Wobj:=Wobj_Part_0;
        Movel Tr_meulage_bavure_122,VitesseRapide,Z0,Tool \Wobj:=Wobj_Part_0;
        Movel Tr_meulage_bavure_123,VitesseRapide,Z0,Tool \Wobj:=Wobj_Part_0;
        Movel Tr_meulage_bavure_124,VitesseRapide,Z0,Tool \Wobj:=Wobj_Part_0;
        Movel Tr_meulage_bavure_125,VitesseRapide,Z0,Tool \Wobj:=Wobj_Part_0;
        Movel Tr_meulage_bavure_126,VitesseRapide,Z0,Tool \Wobj:=Wobj_Part_0;
        Movel Tr_meulage_bavure_127,VitesseRapide,Z0,Tool \Wobj:=Wobj_Part_0;
        Movel Tr_meulage_bavure_128,VitesseRapide,Z0,Tool \Wobj:=Wobj_Part_0;
        Movel Tr_meulage_bavure_129,VitesseRapide,Z0,Tool \Wobj:=Wobj_Part_0;
        Movel Tr_meulage_bavure_130,VitesseRapide,Z0,Tool \Wobj:=Wobj_Part_0;
        Movel Tr_meulage_bavure_131,VitesseRapide,Z0,Tool \Wobj:=Wobj_Part_0;
        Movel Tr_meulage_bavure_132,VitesseRapide,Z0,Tool \Wobj:=Wobj_Part_0;
        Movel Tr_meulage_bavure_133,VitesseRapide,Z0,Tool \Wobj:=Wobj_Part_0;
        Movel Tr_meulage_bavure_134,VitesseRapide,Z0,Tool \Wobj:=Wobj_Part_0;
        Movel Tr_meulage_bavure_135,VitesseRapide,Z0,Tool \Wobj:=Wobj_Part_0;
        Movel Tr_meulage_bavure_136,VitesseRapide,Z0,Tool \Wobj:=Wobj_Part_0;
        Movel Tr_meulage_bavure_137,VitesseRapide,Z0,Tool \Wobj:=Wobj_Part_0;
        Movel Tr_meulage_bavure_138,VitesseRapide,Z0,Tool \Wobj:=Wobj_Part_0;
        Movel Tr_meulage_bavure_139,VitesseRapide,Z0,Tool \Wobj:=Wobj_Part_0;
        Movel Tr_meulage_bavure_140,VitesseRapide,Z0,Tool \Wobj:=Wobj_Part_0;
        Movel Tr_meulage_bavure_141,VitesseRapide,Z0,Tool \Wobj:=Wobj_Part_0;
        Movel Tr_meulage_bavure_142,VitesseRapide,Z0,Tool \Wobj:=Wobj_Part_0;
        Movel Tr_meulage_bavure_143,VitesseRapide,Z0,Tool \Wobj:=Wobj_Part_0;
        Movel Tr_meulage_bavure_144,VitesseRapide,Z0,Tool \Wobj:=Wobj_Part_0;
        Movel Tr_meulage_bavure_145,VitesseRapide,Z0,Tool \Wobj:=Wobj_Part_0;
        Movel Tr_meulage_bavure_146,VitesseRapide,Z0,Tool \Wobj:=Wobj_Part_0;
        Movel Tr_meulage_bavure_147,VitesseRapide,Z0,Tool \Wobj:=Wobj_Part_0;
        Movel Tr_meulage_bavure_148,VitesseRapide,Z0,Tool \Wobj:=Wobj_Part_0;
        Movel Tr_meulage_bavure_149,VitesseRapide,Z0,Tool \Wobj:=Wobj_Part_0;
        Movel Tr_meulage_bavure_150,VitesseRapide,Z0,Tool \Wobj:=Wobj_Part_0;
        Movel Tr_meulage_bavure_151,VitesseRapide,Z0,Tool \Wobj:=Wobj_Part_0;
        Movel Tr_meulage_bavure_152,VitesseRapide,Z0,Tool \Wobj:=Wobj_Part_0;
        Movel Tr_meulage_bavure_153,VitesseRapide,Z0,Tool \Wobj:=Wobj_Part_0;
        Movel Tr_meulage_bavure_154,VitesseRapide,Z0,Tool \Wobj:=Wobj_Part_0;
        Movel Tr_meulage_bavure_155,VitesseRapide,Z0,Tool \Wobj:=Wobj_Part_0;
        Movel Tr_meulage_bavure_156,VitesseRapide,Z0,Tool \Wobj:=Wobj_Part_0;
        Movel Tr_meulage_bavure_157,VitesseRapide,Z0,Tool \Wobj:=Wobj_Part_0;
        Movel Tr_meulage_bavure_158,VitesseRapide,Z0,Tool \Wobj:=Wobj_Part_0;
        Movel Tr_meulage_bavure_159,VitesseRapide,Z0,Tool \Wobj:=Wobj_Part_0;
        Movel Tr_meulage_bavure_160,VitesseRapide,Z0,Tool \Wobj:=Wobj_Part_0;
        Movel Tr_meulage_bavure_161,VitesseRapide,Z0,Tool \Wobj:=Wobj_Part_0;
        Movel Tr_meulage_bavure_162,VitesseRapide,Z0,Tool \Wobj:=Wobj_Part_0;
        Movel Tr_meulage_bavure_163,VitesseRapide,Z0,Tool \Wobj:=Wobj_Part_0;
        Movel Tr_meulage_bavure_164,VitesseRapide,Z0,Tool \Wobj:=Wobj_Part_0;
        Movel Tr_meulage_bavure_165,VitesseRapide,Z0,Tool \Wobj:=Wobj_Part_0;
        Movel Tr_meulage_bavure_166,VitesseRapide,Z0,Tool \Wobj:=Wobj_Part_0;
        Movel Tr_meulage_bavure_167,VitesseRapide,Z0,Tool \Wobj:=Wobj_Part_0;
        Movel Tr_meulage_bavure_168,VitesseRapide,Z0,Tool \Wobj:=Wobj_Part_0;
        Movel Tr_meulage_bavure_169,VitesseRapide,Z0,Tool \Wobj:=Wobj_Part_0;
        Movel Tr_meulage_bavure_170,VitesseRapide,Z0,Tool \Wobj:=Wobj_Part_0;
        Movel Tr_meulage_bavure_171,VitesseRapide,Z0,Tool \Wobj:=Wobj_Part_0;
        Movel Tr_meulage_bavure_172,VitesseRapide,Z0,Tool \Wobj:=Wobj_Part_0;
        Movel Tr_meulage_bavure_173,VitesseRapide,Z0,Tool \Wobj:=Wobj_Part_0;
        Movel Tr_meulage_bavure_174,VitesseRapide,Z0,Tool \Wobj:=Wobj_Part_0;
        Movel Tr_meulage_bavure_175,VitesseRapide,Z0,Tool \Wobj:=Wobj_Part_0;
        Movel Tr_meulage_bavure_176,VitesseRapide,Z0,Tool \Wobj:=Wobj_Part_0;
        Movel Tr_meulage_bavure_177,VitesseRapide,Z0,Tool \Wobj:=Wobj_Part_0;
        Movel Tr_meulage_bavure_178,VitesseRapide,Z0,Tool \Wobj:=Wobj_Part_0;
        Movel Tr_meulage_bavure_179,VitesseRapide,Z0,Tool \Wobj:=Wobj_Part_0;
        Movel Tr_meulage_bavure_180,VitesseRapide,Z0,Tool \Wobj:=Wobj_Part_0;
        Movel Tr_meulage_bavure_181,VitesseRapide,Z0,Tool \Wobj:=Wobj_Part_0;
        Movel Tr_meulage_bavure_182,VitesseRapide,Z0,Tool \Wobj:=Wobj_Part_0;
        Movel Tr_meulage_bavure_183,VitesseRapide,Z0,Tool \Wobj:=Wobj_Part_0;
        Movel Tr_meulage_bavure_184,VitesseRapide,Z0,Tool \Wobj:=Wobj_Part_0;
        Movel Tr_meulage_bavure_185,VitesseRapide,Z0,Tool \Wobj:=Wobj_Part_0;
        Movel Tr_meulage_bavure_186,VitesseRapide,Z0,Tool \Wobj:=Wobj_Part_0;
        Movel Tr_meulage_bavure_187,VitesseRapide,Z0,Tool \Wobj:=Wobj_Part_0;
        Movel Tr_meulage_bavure_188,VitesseRapide,Z0,Tool \Wobj:=Wobj_Part_0;
        Movel Tr_meulage_bavure_189,VitesseRapide,Z0,Tool \Wobj:=Wobj_Part_0;
        Movel Tr_meulage_bavure_190,VitesseRapide,Z0,Tool \Wobj:=Wobj_Part_0;
        Movel Tr_meulage_bavure_191,VitesseRapide,Z0,Tool \Wobj:=Wobj_Part_0;
        Movel Tr_meulage_bavure_192,VitesseRapide,Z0,Tool \Wobj:=Wobj_Part_0;
        Movel Tr_meulage_bavure_193,VitesseRapide,Z0,Tool \Wobj:=Wobj_Part_0;
        Movel Tr_meulage_bavure_194,VitesseRapide,Z0,Tool \Wobj:=Wobj_Part_0;
        Movel Tr_meulage_bavure_195,VitesseRapide,Z0,Tool \Wobj:=Wobj_Part_0;
        Movel Tr_meulage_bavure_196,VitesseRapide,Z0,Tool \Wobj:=Wobj_Part_0;
        Movel Tr_meulage_bavure_197,VitesseRapide,Z0,Tool \Wobj:=Wobj_Part_0;
        Movel Tr_meulage_bavure_198,VitesseRapide,Z0,Tool \Wobj:=Wobj_Part_0;
        Movel Tr_meulage_bavure_199,VitesseRapide,Z0,Tool \Wobj:=Wobj_Part_0;
        Movel Tr_meulage_bavure_200,VitesseRapide,Z0,Tool \Wobj:=Wobj_Part_0;
        Movel Tr_meulage_bavure_201,VitesseRapide,Z0,Tool \Wobj:=Wobj_Part_0;
        Movel Tr_meulage_bavure_202,VitesseRapide,Z0,Tool \Wobj:=Wobj_Part_0;
        Movel Tr_meulage_bavure_203,VitesseRapide,Z0,Tool \Wobj:=Wobj_Part_0;
        Movel Tr_meulage_bavure_204,VitesseRapide,Z0,Tool \Wobj:=Wobj_Part_0;
        Movel Tr_meulage_bavure_205,VitesseRapide,Z0,Tool \Wobj:=Wobj_Part_0;
        Movel Tr_meulage_bavure_206,VitesseRapide,Z0,Tool \Wobj:=Wobj_Part_0;
        Movel Tr_meulage_bavure_207,VitesseRapide,Z0,Tool \Wobj:=Wobj_Part_0;
        Movel Tr_meulage_bavure_208,VitesseRapide,Z0,Tool \Wobj:=Wobj_Part_0;
        Movel Tr_meulage_bavure_209,VitesseRapide,Z0,Tool \Wobj:=Wobj_Part_0;
        Movel Tr_meulage_bavure_210,VitesseRapide,Z0,Tool \Wobj:=Wobj_Part_0;
        Movel Tr_meulage_bavure_211,VitesseRapide,Z0,Tool \Wobj:=Wobj_Part_0;
        Movel Tr_meulage_bavure_212,VitesseRapide,Z0,Tool \Wobj:=Wobj_Part_0;
        Movel Tr_meulage_bavure_213,VitesseRapide,Z0,Tool \Wobj:=Wobj_Part_0;
        Movel Tr_meulage_bavure_214,VitesseRapide,Z0,Tool \Wobj:=Wobj_Part_0;
        Movel Tr_meulage_bavure_215,VitesseRapide,Z0,Tool \Wobj:=Wobj_Part_0;
        Movel Tr_meulage_bavure_216,VitesseRapide,Z0,Tool \Wobj:=Wobj_Part_0;
        Movel Tr_meulage_bavure_217,VitesseRapide,Z0,Tool \Wobj:=Wobj_Part_0;
        Movel Tr_meulage_bavure_218,VitesseRapide,Z0,Tool \Wobj:=Wobj_Part_0;
        Movel Tr_meulage_bavure_219,VitesseRapide,Z0,Tool \Wobj:=Wobj_Part_0;
        Movel Tr_meulage_bavure_220,VitesseRapide,Z0,Tool \Wobj:=Wobj_Part_0;
        Movel Tr_meulage_bavure_221,VitesseRapide,Z0,Tool \Wobj:=Wobj_Part_0;
        Movel Tr_meulage_bavure_222,VitesseRapide,Z0,Tool \Wobj:=Wobj_Part_0;
        Movel Tr_meulage_bavure_223,VitesseRapide,Z0,Tool \Wobj:=Wobj_Part_0;
        Movel Tr_meulage_bavure_224,VitesseRapide,Z0,Tool \Wobj:=Wobj_Part_0;
        Movel Tr_meulage_bavure_225,VitesseRapide,Z0,Tool \Wobj:=Wobj_Part_0;
        Movel Tr_meulage_bavure_226,VitesseRapide,Z0,Tool \Wobj:=Wobj_Part_0;
        Movel Tr_meulage_bavure_227,VitesseRapide,Z0,Tool \Wobj:=Wobj_Part_0;
        Movel Tr_meulage_bavure_228,VitesseRapide,Z0,Tool \Wobj:=Wobj_Part_0;
        Movel Tr_meulage_bavure_229,VitesseRapide,Z0,Tool \Wobj:=Wobj_Part_0;
        Movel Tr_meulage_bavure_230,VitesseRapide,Z0,Tool \Wobj:=Wobj_Part_0;
        Movel Tr_meulage_bavure_231,VitesseRapide,Z0,Tool \Wobj:=Wobj_Part_0;
        Movel Tr_meulage_bavure_232,VitesseRapide,Z0,Tool \Wobj:=Wobj_Part_0;
        Movel Tr_meulage_bavure_233,VitesseRapide,Z0,Tool \Wobj:=Wobj_Part_0;
        Movel Tr_meulage_bavure_234,VitesseRapide,Z0,Tool \Wobj:=Wobj_Part_0;
        Movel Tr_meulage_bavure_235,VitesseRapide,Z0,Tool \Wobj:=Wobj_Part_0;
        Movel Tr_meulage_bavure_236,VitesseRapide,Z0,Tool \Wobj:=Wobj_Part_0;
        Movel Tr_meulage_bavure_237,VitesseRapide,Z0,Tool \Wobj:=Wobj_Part_0;
        Movel Tr_meulage_bavure_238,VitesseRapide,Z0,Tool \Wobj:=Wobj_Part_0;
        Movel Tr_meulage_bavure_239,VitesseRapide,Z0,Tool \Wobj:=Wobj_Part_0;
        Movel Tr_meulage_bavure_240,VitesseRapide,Z0,Tool \Wobj:=Wobj_Part_0;
        Movel Tr_meulage_bavure_241,VitesseRapide,Z0,Tool \Wobj:=Wobj_Part_0;
        Movel Tr_meulage_bavure_242,VitesseRapide,Z0,Tool \Wobj:=Wobj_Part_0;
        Movel Tr_meulage_bavure_243,VitesseRapide,Z0,Tool \Wobj:=Wobj_Part_0;
        Movel Tr_meulage_bavure_244,VitesseRapide,Z0,Tool \Wobj:=Wobj_Part_0;
        Movel Tr_meulage_bavure_245,VitesseRapide,Z0,Tool \Wobj:=Wobj_Part_0;
        Movel Tr_meulage_bavure_246,VitesseRapide,Z0,Tool \Wobj:=Wobj_Part_0;
        Movel Tr_meulage_bavure_247,VitesseRapide,Z0,Tool \Wobj:=Wobj_Part_0;
        Movel Tr_meulage_bavure_248,VitesseRapide,Z0,Tool \Wobj:=Wobj_Part_0;
        Movel Tr_meulage_bavure_249,VitesseRapide,Z0,Tool \Wobj:=Wobj_Part_0;
        Movel Tr_meulage_bavure_250,VitesseRapide,Z0,Tool \Wobj:=Wobj_Part_0;
        Movel Tr_meulage_bavure_251,VitesseRapide,Z0,Tool \Wobj:=Wobj_Part_0;
        Movel Tr_meulage_bavure_252,VitesseRapide,Z0,Tool \Wobj:=Wobj_Part_0;
        Movel Tr_meulage_bavure_253,VitesseRapide,Z0,Tool \Wobj:=Wobj_Part_0;
        Movel Tr_meulage_bavure_254,VitesseRapide,Z0,Tool \Wobj:=Wobj_Part_0;
        Movel Tr_meulage_bavure_255,VitesseRapide,Z0,Tool \Wobj:=Wobj_Part_0;
        Movel Tr_meulage_bavure_256,VitesseRapide,Z0,Tool \Wobj:=Wobj_Part_0;
        Movel Tr_meulage_bavure_257,VitesseRapide,Z0,Tool \Wobj:=Wobj_Part_0;
        Movel Tr_meulage_bavure_258,VitesseRapide,Z0,Tool \Wobj:=Wobj_Part_0;
        Movel Tr_meulage_bavure_259,VitesseRapide,Z0,Tool \Wobj:=Wobj_Part_0;
        Movel Tr_meulage_bavure_260,VitesseRapide,Z0,Tool \Wobj:=Wobj_Part_0;
        Movel Tr_meulage_bavure_261,VitesseRapide,Z0,Tool \Wobj:=Wobj_Part_0;
        Movel Tr_meulage_bavure_262,VitesseRapide,Z0,Tool \Wobj:=Wobj_Part_0;
        Movel Tr_meulage_bavure_263,VitesseRapide,Z0,Tool \Wobj:=Wobj_Part_0;
        Movel Tr_meulage_bavure_264,VitesseRapide,Z0,Tool \Wobj:=Wobj_Part_0;
        Movel Tr_meulage_bavure_265,VitesseRapide,Z0,Tool \Wobj:=Wobj_Part_0;
        Movel Tr_meulage_bavure_266,VitesseRapide,Z0,Tool \Wobj:=Wobj_Part_0;
        Movel Tr_meulage_bavure_267,VitesseRapide,Z0,Tool \Wobj:=Wobj_Part_0;
        Movel Tr_meulage_bavure_268,VitesseRapide,Z0,Tool \Wobj:=Wobj_Part_0;
        Movel Tr_meulage_bavure_269,VitesseRapide,Z0,Tool \Wobj:=Wobj_Part_0;
        Movel Tr_meulage_bavure_270,VitesseRapide,Z0,Tool \Wobj:=Wobj_Part_0;
        Movel Tr_meulage_bavure_271,VitesseRapide,Z0,Tool \Wobj:=Wobj_Part_0;
        Movel Tr_meulage_bavure_272,VitesseRapide,Z0,Tool \Wobj:=Wobj_Part_0;
        Movel Tr_meulage_bavure_273,VitesseRapide,Z0,Tool \Wobj:=Wobj_Part_0;
        Movel Tr_meulage_bavure_274,VitesseRapide,Z0,Tool \Wobj:=Wobj_Part_0;
        Movel Tr_meulage_bavure_275,VitesseRapide,Z0,Tool \Wobj:=Wobj_Part_0;
        Movel Tr_meulage_bavure_276,VitesseRapide,Z0,Tool \Wobj:=Wobj_Part_0;
        Movel Tr_meulage_bavure_277,VitesseRapide,Z0,Tool \Wobj:=Wobj_Part_0;
        Movel Tr_meulage_bavure_278,VitesseRapide,Z0,Tool \Wobj:=Wobj_Part_0;
        Movel Tr_meulage_bavure_279,VitesseRapide,Z0,Tool \Wobj:=Wobj_Part_0;
        Movel Tr_meulage_bavure_280,VitesseRapide,Z0,Tool \Wobj:=Wobj_Part_0;
        Movel Tr_meulage_bavure_281,VitesseRapide,Z0,Tool \Wobj:=Wobj_Part_0;
        Movel Tr_meulage_bavure_282,VitesseRapide,Z0,Tool \Wobj:=Wobj_Part_0;
        Movel Tr_meulage_bavure_283,VitesseRapide,Z0,Tool \Wobj:=Wobj_Part_0;
        Movel Tr_meulage_bavure_284,VitesseRapide,Z0,Tool \Wobj:=Wobj_Part_0;
        Movel Tr_meulage_bavure_285,VitesseRapide,Z0,Tool \Wobj:=Wobj_Part_0;
        Movel Tr_meulage_bavure_286,VitesseRapide,Z0,Tool \Wobj:=Wobj_Part_0;
        Movel Tr_meulage_bavure_287,VitesseRapide,Z0,Tool \Wobj:=Wobj_Part_0;
        Movel Tr_meulage_bavure_288,VitesseRapide,Z0,Tool \Wobj:=Wobj_Part_0;
        Movel Tr_meulage_bavure_289,VitesseRapide,Z0,Tool \Wobj:=Wobj_Part_0;
        Movel Tr_meulage_bavure_290,VitesseRapide,Z0,Tool \Wobj:=Wobj_Part_0;
        Movel Tr_meulage_bavure_291,VitesseRapide,Z0,Tool \Wobj:=Wobj_Part_0;
        Movel Tr_meulage_bavure_292,VitesseRapide,Z0,Tool \Wobj:=Wobj_Part_0;
        Movel Tr_meulage_bavure_293,VitesseRapide,Z0,Tool \Wobj:=Wobj_Part_0;
        Movel Tr_meulage_bavure_294,VitesseRapide,Z0,Tool \Wobj:=Wobj_Part_0;
        Movel Tr_meulage_bavure_295,VitesseRapide,Z0,Tool \Wobj:=Wobj_Part_0;
        Movel Tr_meulage_bavure_296,VitesseRapide,Z0,Tool \Wobj:=Wobj_Part_0;
        Movel Tr_meulage_bavure_297,VitesseRapide,Z0,Tool \Wobj:=Wobj_Part_0;
        Movel Tr_meulage_bavure_298,VitesseRapide,Z0,Tool \Wobj:=Wobj_Part_0;
        Movel Tr_meulage_bavure_299,VitesseRapide,Z0,Tool \Wobj:=Wobj_Part_0;
        Movel Tr_meulage_bavure_300,VitesseRapide,Z0,Tool \Wobj:=Wobj_Part_0;
        Movel Tr_meulage_bavure_301,VitesseRapide,Z0,Tool \Wobj:=Wobj_Part_0;
        Movel Tr_meulage_bavure_302,VitesseRapide,Z0,Tool \Wobj:=Wobj_Part_0;
        Movel Tr_meulage_bavure_303,VitesseRapide,Z0,Tool \Wobj:=Wobj_Part_0;
        Movel Tr_meulage_bavure_304,VitesseRapide,Z0,Tool \Wobj:=Wobj_Part_0;
        Movel Tr_meulage_bavure_305,VitesseRapide,Z0,Tool \Wobj:=Wobj_Part_0;
        Movel Tr_meulage_bavure_306,VitesseRapide,Z0,Tool \Wobj:=Wobj_Part_0;
        Movel Tr_meulage_bavure_307,VitesseRapide,Z0,Tool \Wobj:=Wobj_Part_0;
        Movel Tr_meulage_bavure_308,VitesseRapide,Z0,Tool \Wobj:=Wobj_Part_0;
        Movel Tr_meulage_bavure_309,VitesseRapide,Z0,Tool \Wobj:=Wobj_Part_0;
        Movel Tr_meulage_bavure_310,VitesseRapide,Z0,Tool \Wobj:=Wobj_Part_0;
        Movel Tr_meulage_bavure_311,VitesseRapide,Z0,Tool \Wobj:=Wobj_Part_0;
        Movel Tr_meulage_bavure_312,VitesseRapide,Z0,Tool \Wobj:=Wobj_Part_0;
        Movel Tr_meulage_bavure_313,VitesseRapide,Z0,Tool \Wobj:=Wobj_Part_0;
        Movel Tr_meulage_bavure_314,VitesseRapide,Z0,Tool \Wobj:=Wobj_Part_0;
        Movel Tr_meulage_bavure_315,VitesseRapide,Z0,Tool \Wobj:=Wobj_Part_0;
        Movel Tr_meulage_bavure_316,VitesseRapide,Z0,Tool \Wobj:=Wobj_Part_0;
        Movel Tr_meulage_bavure_317,VitesseRapide,Z0,Tool \Wobj:=Wobj_Part_0;
        Movel Tr_meulage_bavure_318,VitesseRapide,Z0,Tool \Wobj:=Wobj_Part_0;
        Movel Tr_meulage_bavure_319,VitesseRapide,Z0,Tool \Wobj:=Wobj_Part_0;
        Movel Tr_meulage_bavure_320,VitesseRapide,Z0,Tool \Wobj:=Wobj_Part_0;
        Movel Tr_meulage_bavure_321,VitesseRapide,Z0,Tool \Wobj:=Wobj_Part_0;
        Movel Tr_meulage_bavure_322,VitesseRapide,Z0,Tool \Wobj:=Wobj_Part_0;
        Movel Tr_meulage_bavure_323,VitesseRapide,Z0,Tool \Wobj:=Wobj_Part_0;
        Movel Tr_meulage_bavure_324,VitesseRapide,Z0,Tool \Wobj:=Wobj_Part_0;
        Movel Tr_meulage_bavure_325,VitesseRapide,Z0,Tool \Wobj:=Wobj_Part_0;
        Movel Tr_meulage_bavure_326,VitesseRapide,Z0,Tool \Wobj:=Wobj_Part_0;
        Movel Tr_meulage_bavure_327,VitesseRapide,Z0,Tool \Wobj:=Wobj_Part_0;
        Movel Tr_meulage_bavure_328,VitesseRapide,Z0,Tool \Wobj:=Wobj_Part_0;
        Movel Tr_meulage_bavure_329,VitesseRapide,Z0,Tool \Wobj:=Wobj_Part_0;
        Movel Tr_meulage_bavure_330,VitesseRapide,Z0,Tool \Wobj:=Wobj_Part_0;
        Movel Tr_meulage_bavure_331,VitesseRapide,Z0,Tool \Wobj:=Wobj_Part_0;
        Movel Tr_meulage_bavure_332,VitesseRapide,Z0,Tool \Wobj:=Wobj_Part_0;
        Movel Tr_meulage_bavure_333,VitesseRapide,Z0,Tool \Wobj:=Wobj_Part_0;
        Movel Tr_meulage_bavure_334,VitesseRapide,Z0,Tool \Wobj:=Wobj_Part_0;
        Movel Tr_meulage_bavure_335,VitesseRapide,Z0,Tool \Wobj:=Wobj_Part_0;
        Movel Tr_meulage_bavure_336,VitesseRapide,Z0,Tool \Wobj:=Wobj_Part_0;
        Movel Tr_meulage_bavure_337,VitesseRapide,Z0,Tool \Wobj:=Wobj_Part_0;
        Movel Tr_meulage_bavure_338,VitesseRapide,Z0,Tool \Wobj:=Wobj_Part_0;
        Movel Tr_meulage_bavure_339,VitesseRapide,Z0,Tool \Wobj:=Wobj_Part_0;
        Movel Tr_meulage_bavure_340,VitesseRapide,Z0,Tool \Wobj:=Wobj_Part_0;
        Movel Tr_meulage_bavure_341,VitesseRapide,Z0,Tool \Wobj:=Wobj_Part_0;
        Movel Tr_meulage_bavure_342,VitesseRapide,Z0,Tool \Wobj:=Wobj_Part_0;
        Movel Tr_meulage_bavure_343,VitesseRapide,Z0,Tool \Wobj:=Wobj_Part_0;
        Movel Tr_meulage_bavure_344,VitesseRapide,Z0,Tool \Wobj:=Wobj_Part_0;
        Movel Tr_meulage_bavure_345,VitesseRapide,Z0,Tool \Wobj:=Wobj_Part_0;
        Movel Tr_meulage_bavure_346,VitesseRapide,Z0,Tool \Wobj:=Wobj_Part_0;
        Movel Tr_meulage_bavure_347,VitesseRapide,Z0,Tool \Wobj:=Wobj_Part_0;
        Movel Tr_meulage_bavure_348,VitesseRapide,Z0,Tool \Wobj:=Wobj_Part_0;
        Movel Tr_meulage_bavure_349,VitesseRapide,Z0,Tool \Wobj:=Wobj_Part_0;
        Movel Tr_meulage_bavure_350,VitesseRapide,Z0,Tool \Wobj:=Wobj_Part_0;
        Movel Tr_meulage_bavure_351,VitesseRapide,Z0,Tool \Wobj:=Wobj_Part_0;
        Movel Tr_meulage_bavure_352,VitesseRapide,Z0,Tool \Wobj:=Wobj_Part_0;
        Movel Tr_meulage_bavure_353,VitesseRapide,Z0,Tool \Wobj:=Wobj_Part_0;
        Movel Tr_meulage_bavure_354,VitesseRapide,Z0,Tool \Wobj:=Wobj_Part_0;
        Movel Tr_meulage_bavure_355,VitesseRapide,Z0,Tool \Wobj:=Wobj_Part_0;
        Movel Tr_meulage_bavure_356,VitesseRapide,Z0,Tool \Wobj:=Wobj_Part_0;
        Movel Tr_meulage_bavure_357,VitesseRapide,Z0,Tool \Wobj:=Wobj_Part_0;
        Movel Tr_meulage_bavure_358,VitesseRapide,Z0,Tool \Wobj:=Wobj_Part_0;
        Movel Tr_meulage_bavure_359,VitesseRapide,Z0,Tool \Wobj:=Wobj_Part_0;
        Movel Tr_meulage_bavure_360,VitesseRapide,Z0,Tool \Wobj:=Wobj_Part_0;
        Movel Tr_meulage_bavure_361,VitesseRapide,Z0,Tool \Wobj:=Wobj_Part_0;
        Movel Tr_meulage_bavure_362,VitesseRapide,Z0,Tool \Wobj:=Wobj_Part_0;
        Movel Tr_meulage_bavure_363,VitesseRapide,Z0,Tool \Wobj:=Wobj_Part_0;
        Movel Tr_meulage_bavure_364,VitesseRapide,Z0,Tool \Wobj:=Wobj_Part_0;
        Movel Tr_meulage_bavure_365,VitesseRapide,Z0,Tool \Wobj:=Wobj_Part_0;
        Movel Tr_meulage_bavure_366,VitesseRapide,Z0,Tool \Wobj:=Wobj_Part_0;
        Movel Tr_meulage_bavure_367,VitesseRapide,Z0,Tool \Wobj:=Wobj_Part_0;
        Movel Tr_meulage_bavure_368,VitesseRapide,Z0,Tool \Wobj:=Wobj_Part_0;
        Movel Tr_meulage_bavure_369,VitesseRapide,Z0,Tool \Wobj:=Wobj_Part_0;
        Movel Tr_meulage_bavure_370,VitesseRapide,Z0,Tool \Wobj:=Wobj_Part_0;
        Movel Tr_meulage_bavure_371,VitesseRapide,Z0,Tool \Wobj:=Wobj_Part_0;
        Movel Tr_meulage_bavure_372,VitesseRapide,Z0,Tool \Wobj:=Wobj_Part_0;
        Movel Tr_meulage_bavure_373,VitesseRapide,Z0,Tool \Wobj:=Wobj_Part_0;
        Movel Tr_meulage_bavure_374,VitesseRapide,Z0,Tool \Wobj:=Wobj_Part_0;
        Movel Tr_meulage_bavure_375,VitesseRapide,Z0,Tool \Wobj:=Wobj_Part_0;
        Movel Tr_meulage_bavure_376,VitesseRapide,Z0,Tool \Wobj:=Wobj_Part_0;
        Movel Tr_meulage_bavure_377,VitesseRapide,Z0,Tool \Wobj:=Wobj_Part_0;
        Movel Tr_meulage_bavure_378,VitesseRapide,Z0,Tool \Wobj:=Wobj_Part_0;
        Movel Tr_meulage_bavure_379,VitesseRapide,Z0,Tool \Wobj:=Wobj_Part_0;
        Movel Tr_meulage_bavure_380,VitesseRapide,Z0,Tool \Wobj:=Wobj_Part_0;
        Movel Tr_meulage_bavure_381,VitesseRapide,Z0,Tool \Wobj:=Wobj_Part_0;
        Movel Tr_meulage_bavure_382,VitesseRapide,Z0,Tool \Wobj:=Wobj_Part_0;
        Movel Tr_meulage_bavure_383,VitesseRapide,Z0,Tool \Wobj:=Wobj_Part_0;
        Movel Tr_meulage_bavure_384,VitesseRapide,Z0,Tool \Wobj:=Wobj_Part_0;
        Movel Tr_meulage_bavure_385,VitesseRapide,Z0,Tool \Wobj:=Wobj_Part_0;
        Movel Tr_meulage_bavure_386,VitesseRapide,Z0,Tool \Wobj:=Wobj_Part_0;
        Movel Tr_meulage_bavure_387,VitesseRapide,Z0,Tool \Wobj:=Wobj_Part_0;
        Movel Tr_meulage_bavure_388,VitesseRapide,Z0,Tool \Wobj:=Wobj_Part_0;
        Movel Tr_meulage_bavure_389,VitesseRapide,Z0,Tool \Wobj:=Wobj_Part_0;
        Movel Tr_meulage_bavure_390,VitesseRapide,Z0,Tool \Wobj:=Wobj_Part_0;
        Movel Tr_meulage_bavure_391,VitesseRapide,Z0,Tool \Wobj:=Wobj_Part_0;
        Movel Tr_meulage_bavure_392,VitesseRapide,Z0,Tool \Wobj:=Wobj_Part_0;
        Movel Tr_meulage_bavure_393,VitesseRapide,Z0,Tool \Wobj:=Wobj_Part_0;
        Movel Tr_meulage_bavure_394,VitesseRapide,Z0,Tool \Wobj:=Wobj_Part_0;
        Movel Tr_meulage_bavure_395,VitesseRapide,Z0,Tool \Wobj:=Wobj_Part_0;
        Movel Tr_meulage_bavure_396,VitesseRapide,Z0,Tool \Wobj:=Wobj_Part_0;
        Movel Tr_meulage_bavure_397,VitesseRapide,Z0,Tool \Wobj:=Wobj_Part_0;
        Movel Tr_meulage_bavure_398,VitesseRapide,Z0,Tool \Wobj:=Wobj_Part_0;
        Movel Tr_meulage_bavure_399,VitesseRapide,Z0,Tool \Wobj:=Wobj_Part_0;
        Movel Tr_meulage_bavure_400,VitesseRapide,Z0,Tool \Wobj:=Wobj_Part_0;
        Movel Tr_meulage_bavure_401,VitesseRapide,Z0,Tool \Wobj:=Wobj_Part_0;
        Movel Tr_meulage_bavure_402,VitesseRapide,Z0,Tool \Wobj:=Wobj_Part_0;
        Movel Tr_meulage_bavure_403,VitesseRapide,Z0,Tool \Wobj:=Wobj_Part_0;
        Movel Tr_meulage_bavure_404,VitesseRapide,Z0,Tool \Wobj:=Wobj_Part_0;
        Movel Tr_meulage_bavure_405,VitesseRapide,Z0,Tool \Wobj:=Wobj_Part_0;
        Movel Tr_meulage_bavure_406,VitesseRapide,Z0,Tool \Wobj:=Wobj_Part_0;
        Movel Tr_meulage_bavure_407,VitesseRapide,Z0,Tool \Wobj:=Wobj_Part_0;
        Movel Tr_meulage_bavure_408,VitesseRapide,Z0,Tool \Wobj:=Wobj_Part_0;
        Movel Tr_meulage_bavure_409,VitesseRapide,Z0,Tool \Wobj:=Wobj_Part_0;
        Movel Tr_meulage_bavure_410,VitesseRapide,Z0,Tool \Wobj:=Wobj_Part_0;
        Movel Tr_meulage_bavure_411,VitesseRapide,Z0,Tool \Wobj:=Wobj_Part_0;
        Movel Tr_meulage_bavure_412,VitesseRapide,Z0,Tool \Wobj:=Wobj_Part_0;
        Movel Tr_meulage_bavure_413,VitesseRapide,Z0,Tool \Wobj:=Wobj_Part_0;
        Movel Tr_meulage_bavure_414,VitesseRapide,Z0,Tool \Wobj:=Wobj_Part_0;
        Movel Tr_meulage_bavure_415,VitesseRapide,Z0,Tool \Wobj:=Wobj_Part_0;
        Movel Tr_meulage_bavure_416,VitesseRapide,Z0,Tool \Wobj:=Wobj_Part_0;
        Movel Tr_meulage_bavure_417,VitesseRapide,Z0,Tool \Wobj:=Wobj_Part_0;
        Movel Tr_meulage_bavure_418,VitesseRapide,Z0,Tool \Wobj:=Wobj_Part_0;
        Movel Tr_meulage_bavure_419,VitesseRapide,Z0,Tool \Wobj:=Wobj_Part_0;
        Movel Tr_meulage_bavure_420,VitesseRapide,Z0,Tool \Wobj:=Wobj_Part_0;
        Movel Tr_meulage_bavure_421,VitesseRapide,Z0,Tool \Wobj:=Wobj_Part_0;
        Movel Tr_meulage_bavure_422,VitesseRapide,Z0,Tool \Wobj:=Wobj_Part_0;
        Movel Tr_meulage_bavure_423,VitesseRapide,Z0,Tool \Wobj:=Wobj_Part_0;
        Movel Tr_meulage_bavure_424,VitesseRapide,Z0,Tool \Wobj:=Wobj_Part_0;
        Movel Tr_meulage_bavure_425,VitesseRapide,Z0,Tool \Wobj:=Wobj_Part_0;
        Movel Tr_meulage_bavure_426,VitesseRapide,Z0,Tool \Wobj:=Wobj_Part_0;
        Movel Tr_meulage_bavure_427,VitesseRapide,Z0,Tool \Wobj:=Wobj_Part_0;
        Movel Tr_meulage_bavure_428,VitesseRapide,Z0,Tool \Wobj:=Wobj_Part_0;
        Movel Tr_meulage_bavure_429,VitesseRapide,Z0,Tool \Wobj:=Wobj_Part_0;
        Movel Tr_meulage_bavure_430,VitesseRapide,Z0,Tool \Wobj:=Wobj_Part_0;
        Movel Tr_meulage_bavure_431,VitesseRapide,Z0,Tool \Wobj:=Wobj_Part_0;
        Movel Tr_meulage_bavure_432,VitesseRapide,Z0,Tool \Wobj:=Wobj_Part_0;
        Movel Tr_meulage_bavure_433,VitesseRapide,Z0,Tool \Wobj:=Wobj_Part_0;
        Movel Tr_meulage_bavure_434,VitesseRapide,Z0,Tool \Wobj:=Wobj_Part_0;
        Movel Tr_meulage_bavure_435,VitesseRapide,Z0,Tool \Wobj:=Wobj_Part_0;
        Movel Tr_meulage_bavure_436,VitesseRapide,Z0,Tool \Wobj:=Wobj_Part_0;
        Movel Tr_meulage_bavure_437,VitesseRapide,Z0,Tool \Wobj:=Wobj_Part_0;
        Movel Tr_meulage_bavure_438,VitesseRapide,Z0,Tool \Wobj:=Wobj_Part_0;
        Movel Tr_meulage_bavure_439,VitesseRapide,Z0,Tool \Wobj:=Wobj_Part_0;
        Movel Tr_meulage_bavure_440,VitesseRapide,Z0,Tool \Wobj:=Wobj_Part_0;
        Movel Tr_meulage_bavure_441,VitesseRapide,Z0,Tool \Wobj:=Wobj_Part_0;
        Movel Tr_meulage_bavure_442,VitesseRapide,Z0,Tool \Wobj:=Wobj_Part_0;
        Movel Tr_meulage_bavure_443,VitesseRapide,Z0,Tool \Wobj:=Wobj_Part_0;
        Movel Tr_meulage_bavure_444,VitesseRapide,Z0,Tool \Wobj:=Wobj_Part_0;
        Movel Tr_meulage_bavure_445,VitesseRapide,Z0,Tool \Wobj:=Wobj_Part_0;
        Movel Tr_meulage_bavure_446,VitesseRapide,Z0,Tool \Wobj:=Wobj_Part_0;
        Movel Tr_meulage_bavure_447,VitesseRapide,Z0,Tool \Wobj:=Wobj_Part_0;
        Movel Tr_meulage_bavure_448,VitesseRapide,Z0,Tool \Wobj:=Wobj_Part_0;
        Movel Tr_meulage_bavure_449,VitesseRapide,Z0,Tool \Wobj:=Wobj_Part_0;
        Movel Tr_meulage_bavure_450,VitesseRapide,Z0,Tool \Wobj:=Wobj_Part_0;
        Movel Tr_meulage_bavure_451,VitesseRapide,Z0,Tool \Wobj:=Wobj_Part_0;
        Movel Tr_meulage_bavure_452,VitesseRapide,Z0,Tool \Wobj:=Wobj_Part_0;
        Movel Tr_meulage_bavure_453,VitesseRapide,Z0,Tool \Wobj:=Wobj_Part_0;
        Movel Tr_meulage_bavure_454,VitesseRapide,Z0,Tool \Wobj:=Wobj_Part_0;
        Movel Tr_meulage_bavure_455,VitesseRapide,Z0,Tool \Wobj:=Wobj_Part_0;
        Movel Tr_meulage_bavure_456,VitesseRapide,Z0,Tool \Wobj:=Wobj_Part_0;
        Movel Tr_meulage_bavure_457,VitesseRapide,Z0,Tool \Wobj:=Wobj_Part_0;
        Movel Tr_meulage_bavure_458,VitesseRapide,Z0,Tool \Wobj:=Wobj_Part_0;
        Movel Tr_meulage_bavure_459,VitesseRapide,Z0,Tool \Wobj:=Wobj_Part_0;
        Movel Tr_meulage_bavure_460,VitesseRapide,Z0,Tool \Wobj:=Wobj_Part_0;
        Movel Tr_meulage_bavure_461,VitesseRapide,Z0,Tool \Wobj:=Wobj_Part_0;
        Movel Tr_meulage_bavure_462,VitesseRapide,Z0,Tool \Wobj:=Wobj_Part_0;
        !
        !Degagement
        MoveL Reltool(Tr_meulage_bavure_462,0,0,-10),V100,Z0,Tool \Wobj:=Wobj_Part_0;
        MoveL Reltool(Tr_meulage_bavure_462,0,0,-100),V500,Z0,Tool \Wobj:=Wobj_Part_0;
        MoveJ Reltool(Tr_meulage_bavure_462,0,0,-200),V1000,Z0,Tool \Wobj:=Wobj_Part_0;


        Go_to_Meulage_Plan;
        !
        !

    ENDPROC

    !Trajectoire de depose de la piece
    LOCAL PROC DEPOSE()
        !
        stop;

        PEO;

        !
        !Approche
		MoveJ Reltool(PicKPosition,0,0,-200),V1000,Z0,Tool_Prehenseur \Wobj:=Wobj_vision;
		MoveL Reltool(PicKPosition,0,0,-100),V500,Z0,Tool_Prehenseur \Wobj:=Wobj_vision;
		MoveL Reltool(PicKPosition,0,0,-10),V200,Z0,Tool_Prehenseur \Wobj:=Wobj_vision;
		MoveL PicKPosition,V100,Fine,Tool_Prehenseur \Wobj:=Wobj_vision;

        !Fermeture pince
		Gripper_Open;
        !
		MoveL Reltool(PicKPosition,0,0,-200),V500,Z0,Tool_Prehenseur \Wobj:=Wobj_vision;

        !
        PEO;
        !

        !Gripper_Close;

        !
    ENDPROC

ENDMODULE
